LIN{ E6POS: X 712.0875, Y 3.2381, Z -130.0150, A 0, B 90, C 0, E1 0, E2 0, E3 0, E4 0 } C_DIS
LIN{ E6POS: X 712.0906, Y 3.3238, Z -130.0150, A 0, B 90, C 0, E1 0, E2 0, E3 0, E4 0 } C_DIS
LIN{ E6POS: X 712.1099, Y 3.6631, Z -130.0150, A 0, B 90, C 0, E1 0, E2 0, E3 0, E4 0 } C_DIS
LIN{ E6POS: X 712.1445, Y 4.6625, Z -130.0150, A 0, B 90, C 0, E1 0, E2 0, E3 0, E4 0 } C_DIS
LIN{ E6POS: X 712.1475, Y 4.7471, Z -130.0150, A 0, B 90, C 0, E1 0, E2 0, E3 0, E4 0 } C_DIS
LIN{ E6POS: X 712.1666, Y 5.0859, Z -130.0150, A 0, B 90, C 0, E1 0, E2 0, E3 0, E4 0 } C_DIS
LIN{ E6POS: X 712.2006, Y 6.0853, Z -130.0150, A 0, B 90, C 0, E1 0, E2 0, E3 0, E4 0 } C_DIS
LIN{ E6POS: X 712.2023, Y 6.1349, Z -130.0150, A 0, B 90, C 0, E1 0, E2 0, E3 0, E4 0 } C_DIS
LIN{ E6POS: X 712.2215, Y 6.4624, Z -130.0150, A 0, B 90, C 0, E1 0, E2 0, E3 0, E4 0 } C_DIS
LIN{ E6POS: X 712.2546, Y 7.4428, Z -130.0150, A 0, B 90, C 0, E1 0, E2 0, E3 0, E4 0 } C_DIS
LIN{ E6POS: X 712.2745, Y 7.7486, Z -130.0150, A 0, B 90, C 0, E1 0, E2 0, E3 0, E4 0 } C_DIS
LIN{ E6POS: X 712.3050, Y 8.6935, Z -130.0150, A 0, B 90, C 0, E1 0, E2 0, E3 0, E4 0 } C_DIS
LIN{ E6POS: X 712.3249, Y 8.9881, Z -130.0150, A 0, B 90, C 0, E1 0, E2 0, E3 0, E4 0 } C_DIS
LIN{ E6POS: X 712.3556, Y 9.9312, Z -130.0150, A 0, B 90, C 0, E1 0, E2 0, E3 0, E4 0 } C_DIS
LIN{ E6POS: X 712.3754, Y 10.2252, Z -130.0150, A 0, B 90, C 0, E1 0, E2 0, E3 0, E4 0 } C_DIS
LIN{ E6POS: X 712.4064, Y 11.1999, Z -130.0150, A 0, B 90, C 0, E1 0, E2 0, E3 0, E4 0 } C_DIS
LIN{ E6POS: X 712.4258, Y 11.5039, Z -130.0150, A 0, B 90, C 0, E1 0, E2 0, E3 0, E4 0 } C_DIS
LIN{ E6POS: X 712.4588, Y 12.5033, Z -130.0150, A 0, B 90, C 0, E1 0, E2 0, E3 0, E4 0 } C_DIS
LIN{ E6POS: X 712.4601, Y 12.5446, Z -130.0150, A 0, B 90, C 0, E1 0, E2 0, E3 0, E4 0 } C_DIS
LIN{ E6POS: X 712.4786, Y 12.8694, Z -130.0150, A 0, B 90, C 0, E1 0, E2 0, E3 0, E4 0 } C_DIS
LIN{ E6POS: X 712.5115, Y 13.8689, Z -130.0150, A 0, B 90, C 0, E1 0, E2 0, E3 0, E4 0 } C_DIS
LIN{ E6POS: X 712.5138, Y 13.9415, Z -130.0150, A 0, B 90, C 0, E1 0, E2 0, E3 0, E4 0 } C_DIS
LIN{ E6POS: X 712.5317, Y 14.2765, Z -130.0150, A 0, B 90, C 0, E1 0, E2 0, E3 0, E4 0 } C_DIS
LIN{ E6POS: X 712.5651, Y 15.2759, Z -130.0150, A 0, B 90, C 0, E1 0, E2 0, E3 0, E4 0 } C_DIS
LIN{ E6POS: X 712.5675, Y 15.3476, Z -130.0150, A 0, B 90, C 0, E1 0, E2 0, E3 0, E4 0 } C_DIS
LIN{ E6POS: X 712.5857, Y 15.6822, Z -130.0150, A 0, B 90, C 0, E1 0, E2 0, E3 0, E4 0 } C_DIS
LIN{ E6POS: X 712.6192, Y 16.6816, Z -130.0150, A 0, B 90, C 0, E1 0, E2 0, E3 0, E4 0 } C_DIS
LIN{ E6POS: X 712.6205, Y 16.7189, Z -130.0150, A 0, B 90, C 0, E1 0, E2 0, E3 0, E4 0 } C_DIS
LIN{ E6POS: X 712.6389, Y 17.0427, Z -130.0150, A 0, B 90, C 0, E1 0, E2 0, E3 0, E4 0 } C_DIS
LIN{ E6POS: X 712.6716, Y 18.0105, Z -130.0150, A 0, B 90, C 0, E1 0, E2 0, E3 0, E4 0 } C_DIS
LIN{ E6POS: X 712.6913, Y 18.3127, Z -130.0150, A 0, B 90, C 0, E1 0, E2 0, E3 0, E4 0 } C_DIS
LIN{ E6POS: X 712.7222, Y 19.2455, Z -130.0150, A 0, B 90, C 0, E1 0, E2 0, E3 0, E4 0 } C_DIS
LIN{ E6POS: X 712.7422, Y 19.5366, Z -130.0150, A 0, B 90, C 0, E1 0, E2 0, E3 0, E4 0 } C_DIS
LIN{ E6POS: X 712.7740, Y 20.4676, Z -130.0150, A 0, B 90, C 0, E1 0, E2 0, E3 0, E4 0 } C_DIS
LIN{ E6POS: X 712.7943, Y 20.7581, Z -130.0150, A 0, B 90, C 0, E1 0, E2 0, E3 0, E4 0 } C_DIS
LIN{ E6POS: X 712.8292, Y 21.7205, Z -130.0150, A 0, B 90, C 0, E1 0, E2 0, E3 0, E4 0 } C_DIS
LIN{ E6POS: X 712.8492, Y 22.0206, Z -130.0150, A 0, B 90, C 0, E1 0, E2 0, E3 0, E4 0 } C_DIS
LIN{ E6POS: X 712.8860, Y 23.0199, Z -130.0150, A 0, B 90, C 0, E1 0, E2 0, E3 0, E4 0 } C_DIS
LIN{ E6POS: X 712.8870, Y 23.0469, Z -130.0150, A 0, B 90, C 0, E1 0, E2 0, E3 0, E4 0 } C_DIS
LIN{ E6POS: X 712.9064, Y 23.3674, Z -130.0150, A 0, B 90, C 0, E1 0, E2 0, E3 0, E4 0 } C_DIS
LIN{ E6POS: X 712.9477, Y 24.3665, Z -130.0150, A 0, B 90, C 0, E1 0, E2 0, E3 0, E4 0 } C_DIS
LIN{ E6POS: X 712.9490, Y 24.3984, Z -130.0150, A 0, B 90, C 0, E1 0, E2 0, E3 0, E4 0 } C_DIS
LIN{ E6POS: X 712.9686, Y 24.7244, Z -130.0150, A 0, B 90, C 0, E1 0, E2 0, E3 0, E4 0 } C_DIS
LIN{ E6POS: X 713.0131, Y 25.6987, Z -130.0150, A 0, B 90, C 0, E1 0, E2 0, E3 0, E4 0 } C_DIS
LIN{ E6POS: X 713.0333, Y 26.0155, Z -130.0150, A 0, B 90, C 0, E1 0, E2 0, E3 0, E4 0 } C_DIS
LIN{ E6POS: X 713.1012, Y 27.0132, Z -130.0150, A 0, B 90, C 0, E1 0, E2 0, E3 0, E4 0 } C_DIS
LIN{ E6POS: X 713.1591, Y 27.8651, Z -130.0150, A 0, B 90, C 0, E1 0, E2 0, E3 0, E4 0 } C_DIS
LIN{ E6POS: X 713.1805, Y 28.1585, Z -130.0150, A 0, B 90, C 0, E1 0, E2 0, E3 0, E4 0 } C_DIS
LIN{ E6POS: X 713.2037, Y 28.4137, Z -130.0150, A 0, B 90, C 0, E1 0, E2 0, E3 0, E4 0 } C_DIS
LIN{ E6POS: X 713.2279, Y 28.6538, Z -130.0150, A 0, B 90, C 0, E1 0, E2 0, E3 0, E4 0 } C_DIS
LIN{ E6POS: X 713.2526, Y 28.9018, Z -130.0150, A 0, B 90, C 0, E1 0, E2 0, E3 0, E4 0 } C_DIS
LIN{ E6POS: X 713.3221, Y 29.8994, Z -130.0150, A 0, B 90, C 0, E1 0, E2 0, E3 0, E4 0 } C_DIS
LIN{ E6POS: X 713.3798, Y 30.7264, Z -130.0150, A 0, B 90, C 0, E1 0, E2 0, E3 0, E4 0 } C_DIS
LIN{ E6POS: X 713.4036, Y 31.0052, Z -130.0150, A 0, B 90, C 0, E1 0, E2 0, E3 0, E4 0 } C_DIS
LIN{ E6POS: X 713.4446, Y 32.0043, Z -130.0150, A 0, B 90, C 0, E1 0, E2 0, E3 0, E4 0 } C_DIS
LIN{ E6POS: X 713.4495, Y 32.1244, Z -130.0150, A 0, B 90, C 0, E1 0, E2 0, E3 0, E4 0 } C_DIS
LIN{ E6POS: X 713.4719, Y 32.4573, Z -130.0150, A 0, B 90, C 0, E1 0, E2 0, E3 0, E4 0 } C_DIS
LIN{ E6POS: X 713.5074, Y 33.4566, Z -130.0150, A 0, B 90, C 0, E1 0, E2 0, E3 0, E4 0 } C_DIS
LIN{ E6POS: X 713.5167, Y 33.7167, Z -130.0150, A 0, B 90, C 0, E1 0, E2 0, E3 0, E4 0 } C_DIS
LIN{ E6POS: X 713.5383, Y 34.0760, Z -130.0150, A 0, B 90, C 0, E1 0, E2 0, E3 0, E4 0 } C_DIS
LIN{ E6POS: X 713.5743, Y 35.0753, Z -130.0150, A 0, B 90, C 0, E1 0, E2 0, E3 0, E4 0 } C_DIS
LIN{ E6POS: X 713.5836, Y 35.3345, Z -130.0150, A 0, B 90, C 0, E1 0, E2 0, E3 0, E4 0 } C_DIS
LIN{ E6POS: X 713.6057, Y 35.6936, Z -130.0150, A 0, B 90, C 0, E1 0, E2 0, E3 0, E4 0 } C_DIS
LIN{ E6POS: X 713.6489, Y 36.6927, Z -130.0150, A 0, B 90, C 0, E1 0, E2 0, E3 0, E4 0 } C_DIS
LIN{ E6POS: X 713.6541, Y 36.8113, Z -130.0150, A 0, B 90, C 0, E1 0, E2 0, E3 0, E4 0 } C_DIS
LIN{ E6POS: X 713.6775, Y 37.1430, Z -130.0150, A 0, B 90, C 0, E1 0, E2 0, E3 0, E4 0 } C_DIS
LIN{ E6POS: X 713.7518, Y 38.1403, Z -130.0150, A 0, B 90, C 0, E1 0, E2 0, E3 0, E4 0 } C_DIS
LIN{ E6POS: X 713.7913, Y 38.6709, Z -130.0150, A 0, B 90, C 0, E1 0, E2 0, E3 0, E4 0 } C_DIS
LIN{ E6POS: X 713.8170, Y 38.9482, Z -130.0150, A 0, B 90, C 0, E1 0, E2 0, E3 0, E4 0 } C_DIS
LIN{ E6POS: X 713.8444, Y 39.1979, Z -130.0150, A 0, B 90, C 0, E1 0, E2 0, E3 0, E4 0 } C_DIS
LIN{ E6POS: X 713.8728, Y 39.4464, Z -130.0150, A 0, B 90, C 0, E1 0, E2 0, E3 0, E4 0 } C_DIS
LIN{ E6POS: X 713.9560, Y 40.4430, Z -130.0150, A 0, B 90, C 0, E1 0, E2 0, E3 0, E4 0 } C_DIS
LIN{ E6POS: X 713.9993, Y 40.9624, Z -130.0150, A 0, B 90, C 0, E1 0, E2 0, E3 0, E4 0 } C_DIS
LIN{ E6POS: X 714.0283, Y 41.2367, Z -130.0150, A 0, B 90, C 0, E1 0, E2 0, E3 0, E4 0 } C_DIS
LIN{ E6POS: X 714.0908, Y 42.2347, Z -130.0150, A 0, B 90, C 0, E1 0, E2 0, E3 0, E4 0 } C_DIS
LIN{ E6POS: X 714.0971, Y 42.3362, Z -130.0150, A 0, B 90, C 0, E1 0, E2 0, E3 0, E4 0 } C_DIS
LIN{ E6POS: X 714.1256, Y 42.6631, Z -130.0150, A 0, B 90, C 0, E1 0, E2 0, E3 0, E4 0 } C_DIS
LIN{ E6POS: X 714.1815, Y 43.6615, Z -130.0150, A 0, B 90, C 0, E1 0, E2 0, E3 0, E4 0 } C_DIS
LIN{ E6POS: X 714.1964, Y 43.9263, Z -130.0150, A 0, B 90, C 0, E1 0, E2 0, E3 0, E4 0 } C_DIS
LIN{ E6POS: X 714.2252, Y 44.2833, Z -130.0150, A 0, B 90, C 0, E1 0, E2 0, E3 0, E4 0 } C_DIS
LIN{ E6POS: X 714.2796, Y 45.2818, Z -130.0150, A 0, B 90, C 0, E1 0, E2 0, E3 0, E4 0 } C_DIS
LIN{ E6POS: X 714.2967, Y 45.5968, Z -130.0150, A 0, B 90, C 0, E1 0, E2 0, E3 0, E4 0 } C_DIS
LIN{ E6POS: X 714.3259, Y 45.9616, Z -130.0150, A 0, B 90, C 0, E1 0, E2 0, E3 0, E4 0 } C_DIS
LIN{ E6POS: X 714.3828, Y 46.9600, Z -130.0150, A 0, B 90, C 0, E1 0, E2 0, E3 0, E4 0 } C_DIS
LIN{ E6POS: X 714.3973, Y 47.2159, Z -130.0150, A 0, B 90, C 0, E1 0, E2 0, E3 0, E4 0 } C_DIS
LIN{ E6POS: X 714.4272, Y 47.5666, Z -130.0150, A 0, B 90, C 0, E1 0, E2 0, E3 0, E4 0 } C_DIS
LIN{ E6POS: X 714.4923, Y 48.5645, Z -130.0150, A 0, B 90, C 0, E1 0, E2 0, E3 0, E4 0 } C_DIS
LIN{ E6POS: X 714.4978, Y 48.6481, Z -130.0150, A 0, B 90, C 0, E1 0, E2 0, E3 0, E4 0 } C_DIS
LIN{ E6POS: X 714.5287, Y 48.9623, Z -130.0150, A 0, B 90, C 0, E1 0, E2 0, E3 0, E4 0 } C_DIS
LIN{ E6POS: X 714.5991, Y 49.9151, Z -130.0150, A 0, B 90, C 0, E1 0, E2 0, E3 0, E4 0 } C_DIS
LIN{ E6POS: X 714.6305, Y 50.2017, Z -130.0150, A 0, B 90, C 0, E1 0, E2 0, E3 0, E4 0 } C_DIS
LIN{ E6POS: X 714.7003, Y 51.0686, Z -130.0150, A 0, B 90, C 0, E1 0, E2 0, E3 0, E4 0 } C_DIS
LIN{ E6POS: X 714.7325, Y 51.3369, Z -130.0150, A 0, B 90, C 0, E1 0, E2 0, E3 0, E4 0 } C_DIS
LIN{ E6POS: X 714.8029, Y 52.1697, Z -130.0150, A 0, B 90, C 0, E1 0, E2 0, E3 0, E4 0 } C_DIS
LIN{ E6POS: X 714.8884, Y 52.4223, Z -130.0150, A 0, B 90, C 0, E1 0, E2 0, E3 0, E4 0 } C_DIS
LIN{ E6POS: X 715.6198, Y 52.2627, Z -130.0150, A 0, B 90, C 0, E1 0, E2 0, E3 0, E4 0 } C_DIS
LIN{ E6POS: X 716.5857, Y 52.0038, Z -130.0150, A 0, B 90, C 0, E1 0, E2 0, E3 0, E4 0 } C_DIS
LIN{ E6POS: X 717.5516, Y 51.7450, Z -130.0150, A 0, B 90, C 0, E1 0, E2 0, E3 0, E4 0 } C_DIS
LIN{ E6POS: X 717.8004, Y 51.6783, Z -130.0150, A 0, B 90, C 0, E1 0, E2 0, E3 0, E4 0 } C_DIS
LIN{ E6POS: X 718.5842, Y 51.4709, Z -130.0150, A 0, B 90, C 0, E1 0, E2 0, E3 0, E4 0 } C_DIS
LIN{ E6POS: X 719.5486, Y 51.2064, Z -130.0150, A 0, B 90, C 0, E1 0, E2 0, E3 0, E4 0 } C_DIS
LIN{ E6POS: X 720.5129, Y 50.9418, Z -130.0150, A 0, B 90, C 0, E1 0, E2 0, E3 0, E4 0 } C_DIS
LIN{ E6POS: X 721.4773, Y 50.6773, Z -130.0150, A 0, B 90, C 0, E1 0, E2 0, E3 0, E4 0 } C_DIS
LIN{ E6POS: X 722.4417, Y 50.4127, Z -130.0150, A 0, B 90, C 0, E1 0, E2 0, E3 0, E4 0 } C_DIS
LIN{ E6POS: X 722.9421, Y 50.2755, Z -130.0150, A 0, B 90, C 0, E1 0, E2 0, E3 0, E4 0 } C_DIS
LIN{ E6POS: X 723.9022, Y 49.9957, Z -130.0150, A 0, B 90, C 0, E1 0, E2 0, E3 0, E4 0 } C_DIS
LIN{ E6POS: X 724.1924, Y 49.9112, Z -130.0150, A 0, B 90, C 0, E1 0, E2 0, E3 0, E4 0 } C_DIS
LIN{ E6POS: X 725.1562, Y 49.6446, Z -130.0150, A 0, B 90, C 0, E1 0, E2 0, E3 0, E4 0 } C_DIS
LIN{ E6POS: X 726.1200, Y 49.3780, Z -130.0150, A 0, B 90, C 0, E1 0, E2 0, E3 0, E4 0 } C_DIS
LIN{ E6POS: X 727.0838, Y 49.1113, Z -130.0150, A 0, B 90, C 0, E1 0, E2 0, E3 0, E4 0 } C_DIS
LIN{ E6POS: X 728.0476, Y 48.8447, Z -130.0150, A 0, B 90, C 0, E1 0, E2 0, E3 0, E4 0 } C_DIS
LIN{ E6POS: X 729.0114, Y 48.5781, Z -130.0150, A 0, B 90, C 0, E1 0, E2 0, E3 0, E4 0 } C_DIS
LIN{ E6POS: X 729.9752, Y 48.3115, Z -130.0150, A 0, B 90, C 0, E1 0, E2 0, E3 0, E4 0 } C_DIS
LIN{ E6POS: X 730.9390, Y 48.0449, Z -130.0150, A 0, B 90, C 0, E1 0, E2 0, E3 0, E4 0 } C_DIS
LIN{ E6POS: X 731.4545, Y 47.9023, Z -130.0150, A 0, B 90, C 0, E1 0, E2 0, E3 0, E4 0 } C_DIS
LIN{ E6POS: X 732.4135, Y 47.6189, Z -130.0150, A 0, B 90, C 0, E1 0, E2 0, E3 0, E4 0 } C_DIS
LIN{ E6POS: X 733.3725, Y 47.3356, Z -130.0150, A 0, B 90, C 0, E1 0, E2 0, E3 0, E4 0 } C_DIS
LIN{ E6POS: X 733.5370, Y 47.2870, Z -130.0150, A 0, B 90, C 0, E1 0, E2 0, E3 0, E4 0 } C_DIS
LIN{ E6POS: X 734.5038, Y 47.0312, Z -130.0150, A 0, B 90, C 0, E1 0, E2 0, E3 0, E4 0 } C_DIS
LIN{ E6POS: X 735.4705, Y 46.7755, Z -130.0150, A 0, B 90, C 0, E1 0, E2 0, E3 0, E4 0 } C_DIS
LIN{ E6POS: X 736.4372, Y 46.5197, Z -130.0150, A 0, B 90, C 0, E1 0, E2 0, E3 0, E4 0 } C_DIS
LIN{ E6POS: X 737.4040, Y 46.2639, Z -130.0150, A 0, B 90, C 0, E1 0, E2 0, E3 0, E4 0 } C_DIS
LIN{ E6POS: X 738.3707, Y 46.0082, Z -130.0150, A 0, B 90, C 0, E1 0, E2 0, E3 0, E4 0 } C_DIS
LIN{ E6POS: X 739.3374, Y 45.7524, Z -130.0150, A 0, B 90, C 0, E1 0, E2 0, E3 0, E4 0 } C_DIS
LIN{ E6POS: X 740.3042, Y 45.4966, Z -130.0150, A 0, B 90, C 0, E1 0, E2 0, E3 0, E4 0 } C_DIS
LIN{ E6POS: X 741.2709, Y 45.2409, Z -130.0150, A 0, B 90, C 0, E1 0, E2 0, E3 0, E4 0 } C_DIS
LIN{ E6POS: X 742.2377, Y 44.9851, Z -130.0150, A 0, B 90, C 0, E1 0, E2 0, E3 0, E4 0 } C_DIS
LIN{ E6POS: X 742.5361, Y 44.9061, Z -130.0150, A 0, B 90, C 0, E1 0, E2 0, E3 0, E4 0 } C_DIS
LIN{ E6POS: X 743.4986, Y 44.6349, Z -130.0150, A 0, B 90, C 0, E1 0, E2 0, E3 0, E4 0 } C_DIS
LIN{ E6POS: X 744.4611, Y 44.3637, Z -130.0150, A 0, B 90, C 0, E1 0, E2 0, E3 0, E4 0 } C_DIS
LIN{ E6POS: X 745.1256, Y 44.1764, Z -130.0150, A 0, B 90, C 0, E1 0, E2 0, E3 0, E4 0 } C_DIS
LIN{ E6POS: X 746.0978, Y 43.9420, Z -130.0150, A 0, B 90, C 0, E1 0, E2 0, E3 0, E4 0 } C_DIS
LIN{ E6POS: X 747.0699, Y 43.7075, Z -130.0150, A 0, B 90, C 0, E1 0, E2 0, E3 0, E4 0 } C_DIS
LIN{ E6POS: X 748.0420, Y 43.4731, Z -130.0150, A 0, B 90, C 0, E1 0, E2 0, E3 0, E4 0 } C_DIS
LIN{ E6POS: X 749.0142, Y 43.2386, Z -130.0150, A 0, B 90, C 0, E1 0, E2 0, E3 0, E4 0 } C_DIS
LIN{ E6POS: X 749.9863, Y 43.0042, Z -130.0150, A 0, B 90, C 0, E1 0, E2 0, E3 0, E4 0 } C_DIS
LIN{ E6POS: X 750.9584, Y 42.7697, Z -130.0150, A 0, B 90, C 0, E1 0, E2 0, E3 0, E4 0 } C_DIS
LIN{ E6POS: X 751.9305, Y 42.5353, Z -130.0150, A 0, B 90, C 0, E1 0, E2 0, E3 0, E4 0 } C_DIS
LIN{ E6POS: X 752.9027, Y 42.3008, Z -130.0150, A 0, B 90, C 0, E1 0, E2 0, E3 0, E4 0 } C_DIS
LIN{ E6POS: X 753.8748, Y 42.0664, Z -130.0150, A 0, B 90, C 0, E1 0, E2 0, E3 0, E4 0 } C_DIS
LIN{ E6POS: X 754.6995, Y 41.8675, Z -130.0150, A 0, B 90, C 0, E1 0, E2 0, E3 0, E4 0 } C_DIS
LIN{ E6POS: X 755.6683, Y 41.6200, Z -130.0150, A 0, B 90, C 0, E1 0, E2 0, E3 0, E4 0 } C_DIS
LIN{ E6POS: X 756.6372, Y 41.3724, Z -130.0150, A 0, B 90, C 0, E1 0, E2 0, E3 0, E4 0 } C_DIS
LIN{ E6POS: X 757.4699, Y 41.1597, Z -130.0150, A 0, B 90, C 0, E1 0, E2 0, E3 0, E4 0 } C_DIS
LIN{ E6POS: X 758.4505, Y 40.9637, Z -130.0150, A 0, B 90, C 0, E1 0, E2 0, E3 0, E4 0 } C_DIS
LIN{ E6POS: X 759.4311, Y 40.7676, Z -130.0150, A 0, B 90, C 0, E1 0, E2 0, E3 0, E4 0 } C_DIS
LIN{ E6POS: X 760.4117, Y 40.5716, Z -130.0150, A 0, B 90, C 0, E1 0, E2 0, E3 0, E4 0 } C_DIS
LIN{ E6POS: X 761.3923, Y 40.3756, Z -130.0150, A 0, B 90, C 0, E1 0, E2 0, E3 0, E4 0 } C_DIS
LIN{ E6POS: X 762.3729, Y 40.1795, Z -130.0150, A 0, B 90, C 0, E1 0, E2 0, E3 0, E4 0 } C_DIS
LIN{ E6POS: X 763.3535, Y 39.9835, Z -130.0150, A 0, B 90, C 0, E1 0, E2 0, E3 0, E4 0 } C_DIS
LIN{ E6POS: X 764.3340, Y 39.7875, Z -130.0150, A 0, B 90, C 0, E1 0, E2 0, E3 0, E4 0 } C_DIS
LIN{ E6POS: X 765.3146, Y 39.5914, Z -130.0150, A 0, B 90, C 0, E1 0, E2 0, E3 0, E4 0 } C_DIS
LIN{ E6POS: X 766.2952, Y 39.3954, Z -130.0150, A 0, B 90, C 0, E1 0, E2 0, E3 0, E4 0 } C_DIS
LIN{ E6POS: X 766.4520, Y 39.3641, Z -130.0150, A 0, B 90, C 0, E1 0, E2 0, E3 0, E4 0 } C_DIS
LIN{ E6POS: X 767.4308, Y 39.1593, Z -130.0150, A 0, B 90, C 0, E1 0, E2 0, E3 0, E4 0 } C_DIS
LIN{ E6POS: X 768.4096, Y 38.9546, Z -130.0150, A 0, B 90, C 0, E1 0, E2 0, E3 0, E4 0 } C_DIS
LIN{ E6POS: X 769.0778, Y 38.8148, Z -130.0150, A 0, B 90, C 0, E1 0, E2 0, E3 0, E4 0 } C_DIS
LIN{ E6POS: X 770.0711, Y 38.6997, Z -130.0150, A 0, B 90, C 0, E1 0, E2 0, E3 0, E4 0 } C_DIS
LIN{ E6POS: X 771.0645, Y 38.5845, Z -130.0150, A 0, B 90, C 0, E1 0, E2 0, E3 0, E4 0 } C_DIS
LIN{ E6POS: X 772.0578, Y 38.4693, Z -130.0150, A 0, B 90, C 0, E1 0, E2 0, E3 0, E4 0 } C_DIS
LIN{ E6POS: X 773.0512, Y 38.3542, Z -130.0150, A 0, B 90, C 0, E1 0, E2 0, E3 0, E4 0 } C_DIS
LIN{ E6POS: X 774.0445, Y 38.2390, Z -130.0150, A 0, B 90, C 0, E1 0, E2 0, E3 0, E4 0 } C_DIS
LIN{ E6POS: X 775.0379, Y 38.1239, Z -130.0150, A 0, B 90, C 0, E1 0, E2 0, E3 0, E4 0 } C_DIS
LIN{ E6POS: X 776.0312, Y 38.0087, Z -130.0150, A 0, B 90, C 0, E1 0, E2 0, E3 0, E4 0 } C_DIS
LIN{ E6POS: X 776.3033, Y 37.9772, Z -130.0150, A 0, B 90, C 0, E1 0, E2 0, E3 0, E4 0 } C_DIS
LIN{ E6POS: X 777.2964, Y 37.8600, Z -130.0150, A 0, B 90, C 0, E1 0, E2 0, E3 0, E4 0 } C_DIS
LIN{ E6POS: X 778.2895, Y 37.7429, Z -130.0150, A 0, B 90, C 0, E1 0, E2 0, E3 0, E4 0 } C_DIS
LIN{ E6POS: X 778.4588, Y 37.7230, Z -130.0150, A 0, B 90, C 0, E1 0, E2 0, E3 0, E4 0 } C_DIS
LIN{ E6POS: X 779.4586, Y 37.7025, Z -130.0150, A 0, B 90, C 0, E1 0, E2 0, E3 0, E4 0 } C_DIS
LIN{ E6POS: X 780.4584, Y 37.6820, Z -130.0150, A 0, B 90, C 0, E1 0, E2 0, E3 0, E4 0 } C_DIS
LIN{ E6POS: X 781.4582, Y 37.6616, Z -130.0150, A 0, B 90, C 0, E1 0, E2 0, E3 0, E4 0 } C_DIS
LIN{ E6POS: X 782.4579, Y 37.6411, Z -130.0150, A 0, B 90, C 0, E1 0, E2 0, E3 0, E4 0 } C_DIS
LIN{ E6POS: X 783.4577, Y 37.6206, Z -130.0150, A 0, B 90, C 0, E1 0, E2 0, E3 0, E4 0 } C_DIS
LIN{ E6POS: X 784.3674, Y 37.6020, Z -130.0150, A 0, B 90, C 0, E1 0, E2 0, E3 0, E4 0 } C_DIS
LIN{ E6POS: X 785.3672, Y 37.5838, Z -130.0150, A 0, B 90, C 0, E1 0, E2 0, E3 0, E4 0 } C_DIS
LIN{ E6POS: X 786.1700, Y 37.5692, Z -130.0150, A 0, B 90, C 0, E1 0, E2 0, E3 0, E4 0 } C_DIS
LIN{ E6POS: X 787.1675, Y 37.6400, Z -130.0150, A 0, B 90, C 0, E1 0, E2 0, E3 0, E4 0 } C_DIS
LIN{ E6POS: X 788.1650, Y 37.7108, Z -130.0150, A 0, B 90, C 0, E1 0, E2 0, E3 0, E4 0 } C_DIS
LIN{ E6POS: X 789.1625, Y 37.7816, Z -130.0150, A 0, B 90, C 0, E1 0, E2 0, E3 0, E4 0 } C_DIS
LIN{ E6POS: X 790.1600, Y 37.8524, Z -130.0150, A 0, B 90, C 0, E1 0, E2 0, E3 0, E4 0 } C_DIS
LIN{ E6POS: X 791.1575, Y 37.9232, Z -130.0150, A 0, B 90, C 0, E1 0, E2 0, E3 0, E4 0 } C_DIS
LIN{ E6POS: X 791.2008, Y 37.9263, Z -130.0150, A 0, B 90, C 0, E1 0, E2 0, E3 0, E4 0 } C_DIS
LIN{ E6POS: X 792.1981, Y 37.9992, Z -130.0150, A 0, B 90, C 0, E1 0, E2 0, E3 0, E4 0 } C_DIS
LIN{ E6POS: X 792.7685, Y 38.0409, Z -130.0150, A 0, B 90, C 0, E1 0, E2 0, E3 0, E4 0 } C_DIS
LIN{ E6POS: X 793.7601, Y 38.1698, Z -130.0150, A 0, B 90, C 0, E1 0, E2 0, E3 0, E4 0 } C_DIS
LIN{ E6POS: X 794.7518, Y 38.2986, Z -130.0150, A 0, B 90, C 0, E1 0, E2 0, E3 0, E4 0 } C_DIS
LIN{ E6POS: X 795.7435, Y 38.4275, Z -130.0150, A 0, B 90, C 0, E1 0, E2 0, E3 0, E4 0 } C_DIS
LIN{ E6POS: X 796.7351, Y 38.5564, Z -130.0150, A 0, B 90, C 0, E1 0, E2 0, E3 0, E4 0 } C_DIS
LIN{ E6POS: X 797.3598, Y 38.6376, Z -130.0150, A 0, B 90, C 0, E1 0, E2 0, E3 0, E4 0 } C_DIS
LIN{ E6POS: X 798.3514, Y 38.7665, Z -130.0150, A 0, B 90, C 0, E1 0, E2 0, E3 0, E4 0 } C_DIS
LIN{ E6POS: X 798.8097, Y 38.8260, Z -130.0150, A 0, B 90, C 0, E1 0, E2 0, E3 0, E4 0 } C_DIS
LIN{ E6POS: X 798.7068, Y 37.8313, Z -130.0150, A 0, B 90, C 0, E1 0, E2 0, E3 0, E4 0 } C_DIS
LIN{ E6POS: X 798.6040, Y 36.8366, Z -130.0150, A 0, B 90, C 0, E1 0, E2 0, E3 0, E4 0 } C_DIS
LIN{ E6POS: X 798.5012, Y 35.8419, Z -130.0150, A 0, B 90, C 0, E1 0, E2 0, E3 0, E4 0 } C_DIS
LIN{ E6POS: X 798.3983, Y 34.8472, Z -130.0150, A 0, B 90, C 0, E1 0, E2 0, E3 0, E4 0 } C_DIS
LIN{ E6POS: X 798.2955, Y 33.8525, Z -130.0150, A 0, B 90, C 0, E1 0, E2 0, E3 0, E4 0 } C_DIS
LIN{ E6POS: X 798.1927, Y 32.8578, Z -130.0150, A 0, B 90, C 0, E1 0, E2 0, E3 0, E4 0 } C_DIS
LIN{ E6POS: X 798.0898, Y 31.8631, Z -130.0150, A 0, B 90, C 0, E1 0, E2 0, E3 0, E4 0 } C_DIS
LIN{ E6POS: X 797.9870, Y 30.8684, Z -130.0150, A 0, B 90, C 0, E1 0, E2 0, E3 0, E4 0 } C_DIS
LIN{ E6POS: X 797.8842, Y 29.8737, Z -130.0150, A 0, B 90, C 0, E1 0, E2 0, E3 0, E4 0 } C_DIS
LIN{ E6POS: X 797.7813, Y 28.8790, Z -130.0150, A 0, B 90, C 0, E1 0, E2 0, E3 0, E4 0 } C_DIS
LIN{ E6POS: X 797.6785, Y 27.8843, Z -130.0150, A 0, B 90, C 0, E1 0, E2 0, E3 0, E4 0 } C_DIS
LIN{ E6POS: X 797.5757, Y 26.8896, Z -130.0150, A 0, B 90, C 0, E1 0, E2 0, E3 0, E4 0 } C_DIS
LIN{ E6POS: X 797.5273, Y 26.4221, Z -130.0150, A 0, B 90, C 0, E1 0, E2 0, E3 0, E4 0 } C_DIS
LIN{ E6POS: X 797.4245, Y 25.4274, Z -130.0150, A 0, B 90, C 0, E1 0, E2 0, E3 0, E4 0 } C_DIS
LIN{ E6POS: X 797.3217, Y 24.4327, Z -130.0150, A 0, B 90, C 0, E1 0, E2 0, E3 0, E4 0 } C_DIS
LIN{ E6POS: X 797.2188, Y 23.4380, Z -130.0150, A 0, B 90, C 0, E1 0, E2 0, E3 0, E4 0 } C_DIS
LIN{ E6POS: X 797.1224, Y 22.5051, Z -130.0150, A 0, B 90, C 0, E1 0, E2 0, E3 0, E4 0 } C_DIS
LIN{ E6POS: X 797.0002, Y 21.5126, Z -130.0150, A 0, B 90, C 0, E1 0, E2 0, E3 0, E4 0 } C_DIS
LIN{ E6POS: X 796.8780, Y 20.5201, Z -130.0150, A 0, B 90, C 0, E1 0, E2 0, E3 0, E4 0 } C_DIS
LIN{ E6POS: X 796.7559, Y 19.5276, Z -130.0150, A 0, B 90, C 0, E1 0, E2 0, E3 0, E4 0 } C_DIS
LIN{ E6POS: X 796.6337, Y 18.5351, Z -130.0150, A 0, B 90, C 0, E1 0, E2 0, E3 0, E4 0 } C_DIS
LIN{ E6POS: X 796.5115, Y 17.5426, Z -130.0150, A 0, B 90, C 0, E1 0, E2 0, E3 0, E4 0 } C_DIS
LIN{ E6POS: X 796.3893, Y 16.5500, Z -130.0150, A 0, B 90, C 0, E1 0, E2 0, E3 0, E4 0 } C_DIS
LIN{ E6POS: X 796.2672, Y 15.5575, Z -130.0150, A 0, B 90, C 0, E1 0, E2 0, E3 0, E4 0 } C_DIS
LIN{ E6POS: X 796.1450, Y 14.5650, Z -130.0150, A 0, B 90, C 0, E1 0, E2 0, E3 0, E4 0 } C_DIS
LIN{ E6POS: X 796.0228, Y 13.5725, Z -130.0150, A 0, B 90, C 0, E1 0, E2 0, E3 0, E4 0 } C_DIS
LIN{ E6POS: X 795.9006, Y 12.5800, Z -130.0150, A 0, B 90, C 0, E1 0, E2 0, E3 0, E4 0 } C_DIS
LIN{ E6POS: X 795.7785, Y 11.5875, Z -130.0150, A 0, B 90, C 0, E1 0, E2 0, E3 0, E4 0 } C_DIS
LIN{ E6POS: X 795.7041, Y 10.9836, Z -130.0150, A 0, B 90, C 0, E1 0, E2 0, E3 0, E4 0 } C_DIS
LIN{ E6POS: X 795.5819, Y 9.9911, Z -130.0150, A 0, B 90, C 0, E1 0, E2 0, E3 0, E4 0 } C_DIS
LIN{ E6POS: X 795.4598, Y 8.9986, Z -130.0150, A 0, B 90, C 0, E1 0, E2 0, E3 0, E4 0 } C_DIS
LIN{ E6POS: X 795.3376, Y 8.0061, Z -130.0150, A 0, B 90, C 0, E1 0, E2 0, E3 0, E4 0 } C_DIS
LIN{ E6POS: X 795.2562, Y 7.3452, Z -128.0150, A 0, B 90, C 0, E1 0, E2 0, E3 0, E4 0 } C_DIS
LIN{ E6POS: X 795.0854, Y 6.3599, Z -128.0150, A 0, B 90, C 0, E1 0, E2 0, E3 0, E4 0 } C_DIS
LIN{ E6POS: X 794.9146, Y 5.3746, Z -128.0150, A 0, B 90, C 0, E1 0, E2 0, E3 0, E4 0 } C_DIS
LIN{ E6POS: X 794.7438, Y 4.3893, Z -128.0150, A 0, B 90, C 0, E1 0, E2 0, E3 0, E4 0 } C_DIS
LIN{ E6POS: X 794.5730, Y 3.4040, Z -128.0150, A 0, B 90, C 0, E1 0, E2 0, E3 0, E4 0 } C_DIS
LIN{ E6POS: X 794.4021, Y 2.4187, Z -128.0150, A 0, B 90, C 0, E1 0, E2 0, E3 0, E4 0 } C_DIS
LIN{ E6POS: X 794.2313, Y 1.4334, Z -128.0150, A 0, B 90, C 0, E1 0, E2 0, E3 0, E4 0 } C_DIS
LIN{ E6POS: X 794.0605, Y 0.4481, Z -128.0150, A 0, B 90, C 0, E1 0, E2 0, E3 0, E4 0 } C_DIS
LIN{ E6POS: X 793.8897, Y -0.5372, Z -128.0150, A 0, B 90, C 0, E1 0, E2 0, E3 0, E4 0 } C_DIS
LIN{ E6POS: X 793.7189, Y -1.5225, Z -128.0150, A 0, B 90, C 0, E1 0, E2 0, E3 0, E4 0 } C_DIS
LIN{ E6POS: X 793.5481, Y -2.5078, Z -128.0150, A 0, B 90, C 0, E1 0, E2 0, E3 0, E4 0 } C_DIS
LIN{ E6POS: X 793.3871, Y -3.4364, Z -128.0150, A 0, B 90, C 0, E1 0, E2 0, E3 0, E4 0 } C_DIS
LIN{ E6POS: X 793.2162, Y -4.4217, Z -128.0150, A 0, B 90, C 0, E1 0, E2 0, E3 0, E4 0 } C_DIS
LIN{ E6POS: X 793.0454, Y -5.4070, Z -128.0150, A 0, B 90, C 0, E1 0, E2 0, E3 0, E4 0 } C_DIS
LIN{ E6POS: X 793.0310, Y -5.4900, Z -128.0150, A 0, B 90, C 0, E1 0, E2 0, E3 0, E4 0 } C_DIS
LIN{ E6POS: X 792.7476, Y -6.4490, Z -128.0150, A 0, B 90, C 0, E1 0, E2 0, E3 0, E4 0 } C_DIS
LIN{ E6POS: X 792.4642, Y -7.4080, Z -128.0150, A 0, B 90, C 0, E1 0, E2 0, E3 0, E4 0 } C_DIS
LIN{ E6POS: X 792.1808, Y -8.3670, Z -128.0150, A 0, B 90, C 0, E1 0, E2 0, E3 0, E4 0 } C_DIS
LIN{ E6POS: X 791.8974, Y -9.3260, Z -128.0150, A 0, B 90, C 0, E1 0, E2 0, E3 0, E4 0 } C_DIS
LIN{ E6POS: X 791.6139, Y -10.2850, Z -128.0150, A 0, B 90, C 0, E1 0, E2 0, E3 0, E4 0 } C_DIS
LIN{ E6POS: X 791.3305, Y -11.2440, Z -128.0150, A 0, B 90, C 0, E1 0, E2 0, E3 0, E4 0 } C_DIS
LIN{ E6POS: X 791.0471, Y -12.2030, Z -128.0150, A 0, B 90, C 0, E1 0, E2 0, E3 0, E4 0 } C_DIS
LIN{ E6POS: X 790.7637, Y -13.1620, Z -128.0150, A 0, B 90, C 0, E1 0, E2 0, E3 0, E4 0 } C_DIS
LIN{ E6POS: X 790.7102, Y -13.3429, Z -128.0150, A 0, B 90, C 0, E1 0, E2 0, E3 0, E4 0 } C_DIS
LIN{ E6POS: X 790.4268, Y -14.3019, Z -128.0150, A 0, B 90, C 0, E1 0, E2 0, E3 0, E4 0 } C_DIS
LIN{ E6POS: X 790.2681, Y -14.8387, Z -128.0150, A 0, B 90, C 0, E1 0, E2 0, E3 0, E4 0 } C_DIS
LIN{ E6POS: X 789.6733, Y -15.6426, Z -128.0150, A 0, B 90, C 0, E1 0, E2 0, E3 0, E4 0 } C_DIS
LIN{ E6POS: X 789.0784, Y -16.4464, Z -128.0150, A 0, B 90, C 0, E1 0, E2 0, E3 0, E4 0 } C_DIS
LIN{ E6POS: X 788.4835, Y -17.2502, Z -128.0150, A 0, B 90, C 0, E1 0, E2 0, E3 0, E4 0 } C_DIS
LIN{ E6POS: X 787.8887, Y -18.0540, Z -128.0150, A 0, B 90, C 0, E1 0, E2 0, E3 0, E4 0 } C_DIS
LIN{ E6POS: X 787.3452, Y -18.7884, Z -128.0150, A 0, B 90, C 0, E1 0, E2 0, E3 0, E4 0 } C_DIS
LIN{ E6POS: X 786.7884, Y -19.5408, Z -128.0150, A 0, B 90, C 0, E1 0, E2 0, E3 0, E4 0 } C_DIS
LIN{ E6POS: X 785.8324, Y -19.8339, Z -128.0150, A 0, B 90, C 0, E1 0, E2 0, E3 0, E4 0 } C_DIS
LIN{ E6POS: X 784.8763, Y -20.1271, Z -128.0150, A 0, B 90, C 0, E1 0, E2 0, E3 0, E4 0 } C_DIS
LIN{ E6POS: X 783.9202, Y -20.4202, Z -128.0150, A 0, B 90, C 0, E1 0, E2 0, E3 0, E4 0 } C_DIS
LIN{ E6POS: X 783.1205, Y -20.6654, Z -128.0150, A 0, B 90, C 0, E1 0, E2 0, E3 0, E4 0 } C_DIS
LIN{ E6POS: X 782.4311, Y -20.8799, Z -128.0150, A 0, B 90, C 0, E1 0, E2 0, E3 0, E4 0 } C_DIS
LIN{ E6POS: X 781.5918, Y -20.7628, Z -128.0150, A 0, B 90, C 0, E1 0, E2 0, E3 0, E4 0 } C_DIS
LIN{ E6POS: X 780.6009, Y -20.6279, Z -128.0150, A 0, B 90, C 0, E1 0, E2 0, E3 0, E4 0 } C_DIS
LIN{ E6POS: X 779.6100, Y -20.4930, Z -128.0150, A 0, B 90, C 0, E1 0, E2 0, E3 0, E4 0 } C_DIS
LIN{ E6POS: X 778.6192, Y -20.3581, Z -128.0150, A 0, B 90, C 0, E1 0, E2 0, E3 0, E4 0 } C_DIS
LIN{ E6POS: X 777.6283, Y -20.2232, Z -128.0150, A 0, B 90, C 0, E1 0, E2 0, E3 0, E4 0 } C_DIS
LIN{ E6POS: X 777.0370, Y -20.1427, Z -128.0150, A 0, B 90, C 0, E1 0, E2 0, E3 0, E4 0 } C_DIS
LIN{ E6POS: X 776.0649, Y -19.9082, Z -128.0150, A 0, B 90, C 0, E1 0, E2 0, E3 0, E4 0 } C_DIS
LIN{ E6POS: X 776.0296, Y -19.8997, Z -128.0150, A 0, B 90, C 0, E1 0, E2 0, E3 0, E4 0 } C_DIS
LIN{ E6POS: X 775.0551, Y -19.6756, Z -128.0150, A 0, B 90, C 0, E1 0, E2 0, E3 0, E4 0 } C_DIS
LIN{ E6POS: X 774.0805, Y -19.4515, Z -128.0150, A 0, B 90, C 0, E1 0, E2 0, E3 0, E4 0 } C_DIS
LIN{ E6POS: X 773.1059, Y -19.2274, Z -128.0150, A 0, B 90, C 0, E1 0, E2 0, E3 0, E4 0 } C_DIS
LIN{ E6POS: X 772.1313, Y -19.0034, Z -128.0150, A 0, B 90, C 0, E1 0, E2 0, E3 0, E4 0 } C_DIS
LIN{ E6POS: X 771.1568, Y -18.7793, Z -128.0150, A 0, B 90, C 0, E1 0, E2 0, E3 0, E4 0 } C_DIS
LIN{ E6POS: X 770.4461, Y -18.6159, Z -128.0150, A 0, B 90, C 0, E1 0, E2 0, E3 0, E4 0 } C_DIS
LIN{ E6POS: X 769.4553, Y -18.4806, Z -128.0150, A 0, B 90, C 0, E1 0, E2 0, E3 0, E4 0 } C_DIS
LIN{ E6POS: X 769.2531, Y -18.4530, Z -128.0150, A 0, B 90, C 0, E1 0, E2 0, E3 0, E4 0 } C_DIS
LIN{ E6POS: X 768.2612, Y -18.3253, Z -128.0150, A 0, B 90, C 0, E1 0, E2 0, E3 0, E4 0 } C_DIS
LIN{ E6POS: X 767.2694, Y -18.1977, Z -128.0150, A 0, B 90, C 0, E1 0, E2 0, E3 0, E4 0 } C_DIS
LIN{ E6POS: X 766.2776, Y -18.0700, Z -128.0150, A 0, B 90, C 0, E1 0, E2 0, E3 0, E4 0 } C_DIS
LIN{ E6POS: X 765.2858, Y -17.9424, Z -128.0150, A 0, B 90, C 0, E1 0, E2 0, E3 0, E4 0 } C_DIS
LIN{ E6POS: X 764.2940, Y -17.8147, Z -128.0150, A 0, B 90, C 0, E1 0, E2 0, E3 0, E4 0 } C_DIS
LIN{ E6POS: X 763.3021, Y -17.6871, Z -128.0150, A 0, B 90, C 0, E1 0, E2 0, E3 0, E4 0 } C_DIS
LIN{ E6POS: X 762.4979, Y -17.5836, Z -128.0150, A 0, B 90, C 0, E1 0, E2 0, E3 0, E4 0 } C_DIS
LIN{ E6POS: X 761.5004, Y -17.5138, Z -128.0150, A 0, B 90, C 0, E1 0, E2 0, E3 0, E4 0 } C_DIS
LIN{ E6POS: X 761.2573, Y -17.4968, Z -128.0150, A 0, B 90, C 0, E1 0, E2 0, E3 0, E4 0 } C_DIS
LIN{ E6POS: X 760.2595, Y -17.4296, Z -128.0150, A 0, B 90, C 0, E1 0, E2 0, E3 0, E4 0 } C_DIS
LIN{ E6POS: X 759.2618, Y -17.3625, Z -128.0150, A 0, B 90, C 0, E1 0, E2 0, E3 0, E4 0 } C_DIS
LIN{ E6POS: X 758.2640, Y -17.2954, Z -128.0150, A 0, B 90, C 0, E1 0, E2 0, E3 0, E4 0 } C_DIS
LIN{ E6POS: X 757.2663, Y -17.2283, Z -128.0150, A 0, B 90, C 0, E1 0, E2 0, E3 0, E4 0 } C_DIS
LIN{ E6POS: X 756.2685, Y -17.1612, Z -128.0150, A 0, B 90, C 0, E1 0, E2 0, E3 0, E4 0 } C_DIS
LIN{ E6POS: X 755.2708, Y -17.0941, Z -128.0150, A 0, B 90, C 0, E1 0, E2 0, E3 0, E4 0 } C_DIS
LIN{ E6POS: X 754.2730, Y -17.0269, Z -128.0150, A 0, B 90, C 0, E1 0, E2 0, E3 0, E4 0 } C_DIS
LIN{ E6POS: X 754.1553, Y -17.0190, Z -128.0150, A 0, B 90, C 0, E1 0, E2 0, E3 0, E4 0 } C_DIS
LIN{ E6POS: X 753.1554, Y -17.0059, Z -128.0150, A 0, B 90, C 0, E1 0, E2 0, E3 0, E4 0 } C_DIS
LIN{ E6POS: X 753.0051, Y -17.0040, Z -128.0150, A 0, B 90, C 0, E1 0, E2 0, E3 0, E4 0 } C_DIS
LIN{ E6POS: X 752.0053, Y -16.9877, Z -128.0150, A 0, B 90, C 0, E1 0, E2 0, E3 0, E4 0 } C_DIS
LIN{ E6POS: X 751.0054, Y -16.9715, Z -128.0150, A 0, B 90, C 0, E1 0, E2 0, E3 0, E4 0 } C_DIS
LIN{ E6POS: X 750.0055, Y -16.9552, Z -128.0150, A 0, B 90, C 0, E1 0, E2 0, E3 0, E4 0 } C_DIS
LIN{ E6POS: X 749.0057, Y -16.9390, Z -128.0150, A 0, B 90, C 0, E1 0, E2 0, E3 0, E4 0 } C_DIS
LIN{ E6POS: X 748.0058, Y -16.9227, Z -128.0150, A 0, B 90, C 0, E1 0, E2 0, E3 0, E4 0 } C_DIS
LIN{ E6POS: X 747.0059, Y -16.9065, Z -128.0150, A 0, B 90, C 0, E1 0, E2 0, E3 0, E4 0 } C_DIS
LIN{ E6POS: X 746.3792, Y -16.8963, Z -128.0150, A 0, B 90, C 0, E1 0, E2 0, E3 0, E4 0 } C_DIS
LIN{ E6POS: X 745.4575, Y -16.9488, Z -128.0150, A 0, B 90, C 0, E1 0, E2 0, E3 0, E4 0 } C_DIS
LIN{ E6POS: X 744.4585, Y -16.9936, Z -128.0150, A 0, B 90, C 0, E1 0, E2 0, E3 0, E4 0 } C_DIS
LIN{ E6POS: X 743.4595, Y -17.0383, Z -128.0150, A 0, B 90, C 0, E1 0, E2 0, E3 0, E4 0 } C_DIS
LIN{ E6POS: X 742.4605, Y -17.0831, Z -128.0150, A 0, B 90, C 0, E1 0, E2 0, E3 0, E4 0 } C_DIS
LIN{ E6POS: X 741.4615, Y -17.1279, Z -128.0150, A 0, B 90, C 0, E1 0, E2 0, E3 0, E4 0 } C_DIS
LIN{ E6POS: X 740.4625, Y -17.1726, Z -128.0150, A 0, B 90, C 0, E1 0, E2 0, E3 0, E4 0 } C_DIS
LIN{ E6POS: X 740.1320, Y -17.1874, Z -128.0150, A 0, B 90, C 0, E1 0, E2 0, E3 0, E4 0 } C_DIS
LIN{ E6POS: X 739.5768, Y -17.3034, Z -128.0150, A 0, B 90, C 0, E1 0, E2 0, E3 0, E4 0 } C_DIS
LIN{ E6POS: X 738.5919, Y -17.4766, Z -128.0150, A 0, B 90, C 0, E1 0, E2 0, E3 0, E4 0 } C_DIS
LIN{ E6POS: X 737.6070, Y -17.6498, Z -128.0150, A 0, B 90, C 0, E1 0, E2 0, E3 0, E4 0 } C_DIS
LIN{ E6POS: X 736.6221, Y -17.8231, Z -128.0150, A 0, B 90, C 0, E1 0, E2 0, E3 0, E4 0 } C_DIS
LIN{ E6POS: X 736.3745, Y -17.8666, Z -128.0150, A 0, B 90, C 0, E1 0, E2 0, E3 0, E4 0 } C_DIS
LIN{ E6POS: X 736.1866, Y -18.0403, Z -128.0150, A 0, B 90, C 0, E1 0, E2 0, E3 0, E4 0 } C_DIS
LIN{ E6POS: X 735.4082, Y -18.6680, Z -128.0150, A 0, B 90, C 0, E1 0, E2 0, E3 0, E4 0 } C_DIS
LIN{ E6POS: X 735.1104, Y -18.9081, Z -128.0150, A 0, B 90, C 0, E1 0, E2 0, E3 0, E4 0 } C_DIS
LIN{ E6POS: X 735.7832, Y -19.6480, Z -128.0150, A 0, B 90, C 0, E1 0, E2 0, E3 0, E4 0 } C_DIS
LIN{ E6POS: X 736.1620, Y -20.0645, Z -128.0150, A 0, B 90, C 0, E1 0, E2 0, E3 0, E4 0 } C_DIS
LIN{ E6POS: X 736.3423, Y -20.2905, Z -128.0150, A 0, B 90, C 0, E1 0, E2 0, E3 0, E4 0 } C_DIS
LIN{ E6POS: X 737.2548, Y -20.6996, Z -128.0150, A 0, B 90, C 0, E1 0, E2 0, E3 0, E4 0 } C_DIS
LIN{ E6POS: X 738.1673, Y -21.1087, Z -128.0150, A 0, B 90, C 0, E1 0, E2 0, E3 0, E4 0 } C_DIS
LIN{ E6POS: X 739.0797, Y -21.5179, Z -128.0150, A 0, B 90, C 0, E1 0, E2 0, E3 0, E4 0 } C_DIS
LIN{ E6POS: X 739.5226, Y -21.7165, Z -128.0150, A 0, B 90, C 0, E1 0, E2 0, E3 0, E4 0 } C_DIS
LIN{ E6POS: X 740.0716, Y -21.9891, Z -128.0150, A 0, B 90, C 0, E1 0, E2 0, E3 0, E4 0 } C_DIS
LIN{ E6POS: X 741.0252, Y -22.2902, Z -128.0150, A 0, B 90, C 0, E1 0, E2 0, E3 0, E4 0 } C_DIS
LIN{ E6POS: X 741.9788, Y -22.5913, Z -128.0150, A 0, B 90, C 0, E1 0, E2 0, E3 0, E4 0 } C_DIS
LIN{ E6POS: X 742.9324, Y -22.8924, Z -128.0150, A 0, B 90, C 0, E1 0, E2 0, E3 0, E4 0 } C_DIS
LIN{ E6POS: X 743.8860, Y -23.1935, Z -128.0150, A 0, B 90, C 0, E1 0, E2 0, E3 0, E4 0 } C_DIS
LIN{ E6POS: X 744.8396, Y -23.4946, Z -128.0150, A 0, B 90, C 0, E1 0, E2 0, E3 0, E4 0 } C_DIS
LIN{ E6POS: X 745.3831, Y -23.6662, Z -128.0150, A 0, B 90, C 0, E1 0, E2 0, E3 0, E4 0 } C_DIS
LIN{ E6POS: X 746.3019, Y -23.9800, Z -128.0150, A 0, B 90, C 0, E1 0, E2 0, E3 0, E4 0 } C_DIS
LIN{ E6POS: X 747.2712, Y -24.2258, Z -128.0150, A 0, B 90, C 0, E1 0, E2 0, E3 0, E4 0 } C_DIS
LIN{ E6POS: X 748.2405, Y -24.4715, Z -128.0150, A 0, B 90, C 0, E1 0, E2 0, E3 0, E4 0 } C_DIS
LIN{ E6POS: X 749.2099, Y -24.7173, Z -128.0150, A 0, B 90, C 0, E1 0, E2 0, E3 0, E4 0 } C_DIS
LIN{ E6POS: X 750.1792, Y -24.9631, Z -128.0150, A 0, B 90, C 0, E1 0, E2 0, E3 0, E4 0 } C_DIS
LIN{ E6POS: X 751.1485, Y -25.2088, Z -128.0150, A 0, B 90, C 0, E1 0, E2 0, E3 0, E4 0 } C_DIS
LIN{ E6POS: X 752.1179, Y -25.4546, Z -128.0150, A 0, B 90, C 0, E1 0, E2 0, E3 0, E4 0 } C_DIS
LIN{ E6POS: X 752.9210, Y -25.6582, Z -128.0150, A 0, B 90, C 0, E1 0, E2 0, E3 0, E4 0 } C_DIS
LIN{ E6POS: X 753.8865, Y -25.9185, Z -128.0150, A 0, B 90, C 0, E1 0, E2 0, E3 0, E4 0 } C_DIS
LIN{ E6POS: X 754.0706, Y -25.9681, Z -128.0150, A 0, B 90, C 0, E1 0, E2 0, E3 0, E4 0 } C_DIS
LIN{ E6POS: X 755.0510, Y -26.1653, Z -128.0150, A 0, B 90, C 0, E1 0, E2 0, E3 0, E4 0 } C_DIS
LIN{ E6POS: X 756.0314, Y -26.3625, Z -128.0150, A 0, B 90, C 0, E1 0, E2 0, E3 0, E4 0 } C_DIS
LIN{ E6POS: X 757.0117, Y -26.5597, Z -128.0150, A 0, B 90, C 0, E1 0, E2 0, E3 0, E4 0 } C_DIS
LIN{ E6POS: X 757.9921, Y -26.7569, Z -128.0150, A 0, B 90, C 0, E1 0, E2 0, E3 0, E4 0 } C_DIS
LIN{ E6POS: X 758.9724, Y -26.9541, Z -128.0150, A 0, B 90, C 0, E1 0, E2 0, E3 0, E4 0 } C_DIS
LIN{ E6POS: X 759.9528, Y -27.1513, Z -128.0150, A 0, B 90, C 0, E1 0, E2 0, E3 0, E4 0 } C_DIS
LIN{ E6POS: X 760.9332, Y -27.3485, Z -128.0150, A 0, B 90, C 0, E1 0, E2 0, E3 0, E4 0 } C_DIS
LIN{ E6POS: X 761.1718, Y -27.3965, Z -128.0150, A 0, B 90, C 0, E1 0, E2 0, E3 0, E4 0 } C_DIS
LIN{ E6POS: X 762.1504, Y -27.6022, Z -128.0150, A 0, B 90, C 0, E1 0, E2 0, E3 0, E4 0 } C_DIS
LIN{ E6POS: X 762.4137, Y -27.6575, Z -128.0150, A 0, B 90, C 0, E1 0, E2 0, E3 0, E4 0 } C_DIS
LIN{ E6POS: X 763.4044, Y -27.7935, Z -128.0150, A 0, B 90, C 0, E1 0, E2 0, E3 0, E4 0 } C_DIS
LIN{ E6POS: X 764.3951, Y -27.9295, Z -128.0150, A 0, B 90, C 0, E1 0, E2 0, E3 0, E4 0 } C_DIS
LIN{ E6POS: X 765.3858, Y -28.0655, Z -128.0150, A 0, B 90, C 0, E1 0, E2 0, E3 0, E4 0 } C_DIS
LIN{ E6POS: X 766.3766, Y -28.2014, Z -128.0150, A 0, B 90, C 0, E1 0, E2 0, E3 0, E4 0 } C_DIS
LIN{ E6POS: X 767.3673, Y -28.3374, Z -128.0150, A 0, B 90, C 0, E1 0, E2 0, E3 0, E4 0 } C_DIS
LIN{ E6POS: X 768.3580, Y -28.4734, Z -128.0150, A 0, B 90, C 0, E1 0, E2 0, E3 0, E4 0 } C_DIS
LIN{ E6POS: X 769.1744, Y -28.5854, Z -128.0150, A 0, B 90, C 0, E1 0, E2 0, E3 0, E4 0 } C_DIS
LIN{ E6POS: X 770.1648, Y -28.7238, Z -128.0150, A 0, B 90, C 0, E1 0, E2 0, E3 0, E4 0 } C_DIS
LIN{ E6POS: X 770.3698, Y -28.7524, Z -128.0150, A 0, B 90, C 0, E1 0, E2 0, E3 0, E4 0 } C_DIS
LIN{ E6POS: X 771.3693, Y -28.7841, Z -128.0150, A 0, B 90, C 0, E1 0, E2 0, E3 0, E4 0 } C_DIS
LIN{ E6POS: X 772.3688, Y -28.8158, Z -128.0150, A 0, B 90, C 0, E1 0, E2 0, E3 0, E4 0 } C_DIS
LIN{ E6POS: X 773.3683, Y -28.8475, Z -128.0150, A 0, B 90, C 0, E1 0, E2 0, E3 0, E4 0 } C_DIS
LIN{ E6POS: X 774.3678, Y -28.8792, Z -128.0150, A 0, B 90, C 0, E1 0, E2 0, E3 0, E4 0 } C_DIS
LIN{ E6POS: X 775.3673, Y -28.9109, Z -128.0150, A 0, B 90, C 0, E1 0, E2 0, E3 0, E4 0 } C_DIS
LIN{ E6POS: X 775.9642, Y -28.9298, Z -128.0150, A 0, B 90, C 0, E1 0, E2 0, E3 0, E4 0 } C_DIS
LIN{ E6POS: X 776.9638, Y -28.9573, Z -128.0150, A 0, B 90, C 0, E1 0, E2 0, E3 0, E4 0 } C_DIS
LIN{ E6POS: X 776.9745, Y -28.9576, Z -128.0150, A 0, B 90, C 0, E1 0, E2 0, E3 0, E4 0 } C_DIS
LIN{ E6POS: X 777.9572, Y -29.1432, Z -128.0150, A 0, B 90, C 0, E1 0, E2 0, E3 0, E4 0 } C_DIS
LIN{ E6POS: X 778.9398, Y -29.3289, Z -128.0150, A 0, B 90, C 0, E1 0, E2 0, E3 0, E4 0 } C_DIS
LIN{ E6POS: X 779.9224, Y -29.5145, Z -128.0150, A 0, B 90, C 0, E1 0, E2 0, E3 0, E4 0 } C_DIS
LIN{ E6POS: X 780.9050, Y -29.7001, Z -128.0150, A 0, B 90, C 0, E1 0, E2 0, E3 0, E4 0 } C_DIS
LIN{ E6POS: X 781.2002, Y -29.7558, Z -128.0150, A 0, B 90, C 0, E1 0, E2 0, E3 0, E4 0 } C_DIS
LIN{ E6POS: X 781.9775, Y -29.9049, Z -128.0150, A 0, B 90, C 0, E1 0, E2 0, E3 0, E4 0 } C_DIS
LIN{ E6POS: X 782.6666, Y -30.6295, Z -128.0150, A 0, B 90, C 0, E1 0, E2 0, E3 0, E4 0 } C_DIS
LIN{ E6POS: X 783.3558, Y -31.3541, Z -128.0150, A 0, B 90, C 0, E1 0, E2 0, E3 0, E4 0 } C_DIS
LIN{ E6POS: X 784.0449, Y -32.0788, Z -128.0150, A 0, B 90, C 0, E1 0, E2 0, E3 0, E4 0 } C_DIS
LIN{ E6POS: X 784.6318, Y -32.6959, Z -128.0150, A 0, B 90, C 0, E1 0, E2 0, E3 0, E4 0 } C_DIS
LIN{ E6POS: X 785.1281, Y -33.2266, Z -128.0150, A 0, B 90, C 0, E1 0, E2 0, E3 0, E4 0 } C_DIS
LIN{ E6POS: X 785.2695, Y -34.2166, Z -128.0150, A 0, B 90, C 0, E1 0, E2 0, E3 0, E4 0 } C_DIS
LIN{ E6POS: X 785.4109, Y -35.2065, Z -128.0150, A 0, B 90, C 0, E1 0, E2 0, E3 0, E4 0 } C_DIS
LIN{ E6POS: X 785.5523, Y -36.1965, Z -128.0150, A 0, B 90, C 0, E1 0, E2 0, E3 0, E4 0 } C_DIS
LIN{ E6POS: X 785.6937, Y -37.1864, Z -128.0150, A 0, B 90, C 0, E1 0, E2 0, E3 0, E4 0 } C_DIS
LIN{ E6POS: X 785.8351, Y -38.1764, Z -128.0150, A 0, B 90, C 0, E1 0, E2 0, E3 0, E4 0 } C_DIS
LIN{ E6POS: X 785.9765, Y -39.1663, Z -128.0150, A 0, B 90, C 0, E1 0, E2 0, E3 0, E4 0 } C_DIS
LIN{ E6POS: X 786.0072, Y -39.3813, Z -128.0150, A 0, B 90, C 0, E1 0, E2 0, E3 0, E4 0 } C_DIS
LIN{ E6POS: X 786.1486, Y -40.3712, Z -128.0150, A 0, B 90, C 0, E1 0, E2 0, E3 0, E4 0 } C_DIS
LIN{ E6POS: X 786.1747, Y -40.5536, Z -128.0150, A 0, B 90, C 0, E1 0, E2 0, E3 0, E4 0 } C_DIS
LIN{ E6POS: X 786.0743, Y -41.5485, Z -128.0150, A 0, B 90, C 0, E1 0, E2 0, E3 0, E4 0 } C_DIS
LIN{ E6POS: X 785.9740, Y -42.5435, Z -128.0150, A 0, B 90, C 0, E1 0, E2 0, E3 0, E4 0 } C_DIS
LIN{ E6POS: X 785.8737, Y -43.5384, Z -128.0150, A 0, B 90, C 0, E1 0, E2 0, E3 0, E4 0 } C_DIS
LIN{ E6POS: X 785.7734, Y -44.5334, Z -128.0150, A 0, B 90, C 0, E1 0, E2 0, E3 0, E4 0 } C_DIS
LIN{ E6POS: X 785.6731, Y -45.5283, Z -128.0150, A 0, B 90, C 0, E1 0, E2 0, E3 0, E4 0 } C_DIS
LIN{ E6POS: X 785.5728, Y -46.5233, Z -128.0150, A 0, B 90, C 0, E1 0, E2 0, E3 0, E4 0 } C_DIS
LIN{ E6POS: X 785.4725, Y -47.5183, Z -128.0150, A 0, B 90, C 0, E1 0, E2 0, E3 0, E4 0 } C_DIS
LIN{ E6POS: X 785.3721, Y -48.5132, Z -128.0150, A 0, B 90, C 0, E1 0, E2 0, E3 0, E4 0 } C_DIS
LIN{ E6POS: X 785.2718, Y -49.5082, Z -128.0150, A 0, B 90, C 0, E1 0, E2 0, E3 0, E4 0 } C_DIS
LIN{ E6POS: X 785.1715, Y -50.5031, Z -128.0150, A 0, B 90, C 0, E1 0, E2 0, E3 0, E4 0 } C_DIS
LIN{ E6POS: X 785.0766, Y -51.4441, Z -128.0150, A 0, B 90, C 0, E1 0, E2 0, E3 0, E4 0 } C_DIS
LIN{ E6POS: X 784.9763, Y -52.4390, Z -128.0150, A 0, B 90, C 0, E1 0, E2 0, E3 0, E4 0 } C_DIS
LIN{ E6POS: X 784.8760, Y -53.4340, Z -128.0150, A 0, B 90, C 0, E1 0, E2 0, E3 0, E4 0 } C_DIS
LIN{ E6POS: X 784.8675, Y -53.5185, Z -128.0150, A 0, B 90, C 0, E1 0, E2 0, E3 0, E4 0 } C_DIS
LIN{ E6POS: X 784.6915, Y -54.5029, Z -128.0150, A 0, B 90, C 0, E1 0, E2 0, E3 0, E4 0 } C_DIS
LIN{ E6POS: X 784.5156, Y -55.4873, Z -128.0150, A 0, B 90, C 0, E1 0, E2 0, E3 0, E4 0 } C_DIS
LIN{ E6POS: X 784.3396, Y -56.4717, Z -128.0150, A 0, B 90, C 0, E1 0, E2 0, E3 0, E4 0 } C_DIS
LIN{ E6POS: X 784.1637, Y -57.4560, Z -128.0150, A 0, B 90, C 0, E1 0, E2 0, E3 0, E4 0 } C_DIS
LIN{ E6POS: X 783.9877, Y -58.4404, Z -128.0150, A 0, B 90, C 0, E1 0, E2 0, E3 0, E4 0 } C_DIS
LIN{ E6POS: X 783.8118, Y -59.4248, Z -128.0150, A 0, B 90, C 0, E1 0, E2 0, E3 0, E4 0 } C_DIS
LIN{ E6POS: X 783.6358, Y -60.4092, Z -128.0150, A 0, B 90, C 0, E1 0, E2 0, E3 0, E4 0 } C_DIS
LIN{ E6POS: X 783.4599, Y -61.3936, Z -128.0150, A 0, B 90, C 0, E1 0, E2 0, E3 0, E4 0 } C_DIS
LIN{ E6POS: X 783.2839, Y -62.3780, Z -128.0150, A 0, B 90, C 0, E1 0, E2 0, E3 0, E4 0 } C_DIS
LIN{ E6POS: X 783.1080, Y -63.3624, Z -128.0150, A 0, B 90, C 0, E1 0, E2 0, E3 0, E4 0 } C_DIS
LIN{ E6POS: X 782.9320, Y -64.3468, Z -128.0150, A 0, B 90, C 0, E1 0, E2 0, E3 0, E4 0 } C_DIS
LIN{ E6POS: X 782.7561, Y -65.3312, Z -128.0150, A 0, B 90, C 0, E1 0, E2 0, E3 0, E4 0 } C_DIS
LIN{ E6POS: X 782.5801, Y -66.3156, Z -128.0150, A 0, B 90, C 0, E1 0, E2 0, E3 0, E4 0 } C_DIS
LIN{ E6POS: X 782.4042, Y -67.3000, Z -128.0150, A 0, B 90, C 0, E1 0, E2 0, E3 0, E4 0 } C_DIS
LIN{ E6POS: X 782.2861, Y -67.9609, Z -128.0150, A 0, B 90, C 0, E1 0, E2 0, E3 0, E4 0 } C_DIS
LIN{ E6POS: X 782.1101, Y -68.9453, Z -128.0150, A 0, B 90, C 0, E1 0, E2 0, E3 0, E4 0 } C_DIS
LIN{ E6POS: X 781.9341, Y -69.9297, Z -128.0150, A 0, B 90, C 0, E1 0, E2 0, E3 0, E4 0 } C_DIS
LIN{ E6POS: X 781.7943, Y -70.7119, Z -128.0150, A 0, B 90, C 0, E1 0, E2 0, E3 0, E4 0 } C_DIS
LIN{ E6POS: X 781.5865, Y -71.6900, Z -128.0150, A 0, B 90, C 0, E1 0, E2 0, E3 0, E4 0 } C_DIS
LIN{ E6POS: X 781.3787, Y -72.6682, Z -128.0150, A 0, B 90, C 0, E1 0, E2 0, E3 0, E4 0 } C_DIS
LIN{ E6POS: X 781.1709, Y -73.6464, Z -128.0150, A 0, B 90, C 0, E1 0, E2 0, E3 0, E4 0 } C_DIS
LIN{ E6POS: X 780.9631, Y -74.6245, Z -128.0150, A 0, B 90, C 0, E1 0, E2 0, E3 0, E4 0 } C_DIS
LIN{ E6POS: X 780.7553, Y -75.6027, Z -128.0150, A 0, B 90, C 0, E1 0, E2 0, E3 0, E4 0 } C_DIS
LIN{ E6POS: X 780.5475, Y -76.5809, Z -128.0150, A 0, B 90, C 0, E1 0, E2 0, E3 0, E4 0 } C_DIS
LIN{ E6POS: X 780.3397, Y -77.5590, Z -128.0150, A 0, B 90, C 0, E1 0, E2 0, E3 0, E4 0 } C_DIS
LIN{ E6POS: X 780.1319, Y -78.5372, Z -128.0150, A 0, B 90, C 0, E1 0, E2 0, E3 0, E4 0 } C_DIS
LIN{ E6POS: X 779.9241, Y -79.5154, Z -128.0150, A 0, B 90, C 0, E1 0, E2 0, E3 0, E4 0 } C_DIS
LIN{ E6POS: X 779.7163, Y -80.4936, Z -128.0150, A 0, B 90, C 0, E1 0, E2 0, E3 0, E4 0 } C_DIS
LIN{ E6POS: X 779.5085, Y -81.4717, Z -128.0150, A 0, B 90, C 0, E1 0, E2 0, E3 0, E4 0 } C_DIS
LIN{ E6POS: X 779.3007, Y -82.4499, Z -128.0150, A 0, B 90, C 0, E1 0, E2 0, E3 0, E4 0 } C_DIS
LIN{ E6POS: X 779.0929, Y -83.4281, Z -128.0150, A 0, B 90, C 0, E1 0, E2 0, E3 0, E4 0 } C_DIS
LIN{ E6POS: X 778.8851, Y -84.4062, Z -128.0150, A 0, B 90, C 0, E1 0, E2 0, E3 0, E4 0 } C_DIS
LIN{ E6POS: X 778.6773, Y -85.3844, Z -128.0150, A 0, B 90, C 0, E1 0, E2 0, E3 0, E4 0 } C_DIS
LIN{ E6POS: X 778.4695, Y -86.3626, Z -128.0150, A 0, B 90, C 0, E1 0, E2 0, E3 0, E4 0 } C_DIS
LIN{ E6POS: X 778.2617, Y -87.3408, Z -128.0150, A 0, B 90, C 0, E1 0, E2 0, E3 0, E4 0 } C_DIS
LIN{ E6POS: X 778.2231, Y -87.5223, Z -128.0150, A 0, B 90, C 0, E1 0, E2 0, E3 0, E4 0 } C_DIS
LIN{ E6POS: X 778.0153, Y -88.5005, Z -128.0150, A 0, B 90, C 0, E1 0, E2 0, E3 0, E4 0 } C_DIS
LIN{ E6POS: X 777.8075, Y -89.4786, Z -128.0150, A 0, B 90, C 0, E1 0, E2 0, E3 0, E4 0 } C_DIS
LIN{ E6POS: X 777.5997, Y -90.4568, Z -128.0150, A 0, B 90, C 0, E1 0, E2 0, E3 0, E4 0 } C_DIS
LIN{ E6POS: X 777.5429, Y -90.7243, Z -128.0150, A 0, B 90, C 0, E1 0, E2 0, E3 0, E4 0 } C_DIS
LIN{ E6POS: X 777.3226, Y -91.6997, Z -128.0150, A 0, B 90, C 0, E1 0, E2 0, E3 0, E4 0 } C_DIS
LIN{ E6POS: X 777.1022, Y -92.6751, Z -128.0150, A 0, B 90, C 0, E1 0, E2 0, E3 0, E4 0 } C_DIS
LIN{ E6POS: X 776.8819, Y -93.6506, Z -128.0150, A 0, B 90, C 0, E1 0, E2 0, E3 0, E4 0 } C_DIS
LIN{ E6POS: X 776.6615, Y -94.6260, Z -128.0150, A 0, B 90, C 0, E1 0, E2 0, E3 0, E4 0 } C_DIS
LIN{ E6POS: X 776.4412, Y -95.6014, Z -128.0150, A 0, B 90, C 0, E1 0, E2 0, E3 0, E4 0 } C_DIS
LIN{ E6POS: X 776.2208, Y -96.5768, Z -128.0150, A 0, B 90, C 0, E1 0, E2 0, E3 0, E4 0 } C_DIS
LIN{ E6POS: X 776.0005, Y -97.5522, Z -128.0150, A 0, B 90, C 0, E1 0, E2 0, E3 0, E4 0 } C_DIS
LIN{ E6POS: X 775.7802, Y -98.5277, Z -128.0150, A 0, B 90, C 0, E1 0, E2 0, E3 0, E4 0 } C_DIS
LIN{ E6POS: X 775.5598, Y -99.5031, Z -128.0150, A 0, B 90, C 0, E1 0, E2 0, E3 0, E4 0 } C_DIS
LIN{ E6POS: X 775.3395, Y -100.4785, Z -128.0150, A 0, B 90, C 0, E1 0, E2 0, E3 0, E4 0 } C_DIS
LIN{ E6POS: X 775.1191, Y -101.4539, Z -128.0150, A 0, B 90, C 0, E1 0, E2 0, E3 0, E4 0 } C_DIS
LIN{ E6POS: X 774.8988, Y -102.4294, Z -128.0150, A 0, B 90, C 0, E1 0, E2 0, E3 0, E4 0 } C_DIS
LIN{ E6POS: X 774.6784, Y -103.4048, Z -128.0150, A 0, B 90, C 0, E1 0, E2 0, E3 0, E4 0 } C_DIS
LIN{ E6POS: X 774.4581, Y -104.3802, Z -128.0150, A 0, B 90, C 0, E1 0, E2 0, E3 0, E4 0 } C_DIS
LIN{ E6POS: X 774.2377, Y -105.3556, Z -128.0150, A 0, B 90, C 0, E1 0, E2 0, E3 0, E4 0 } C_DIS
LIN{ E6POS: X 774.0174, Y -106.3310, Z -128.0150, A 0, B 90, C 0, E1 0, E2 0, E3 0, E4 0 } C_DIS
LIN{ E6POS: X 773.7970, Y -107.3065, Z -128.0150, A 0, B 90, C 0, E1 0, E2 0, E3 0, E4 0 } C_DIS
LIN{ E6POS: X 773.5767, Y -108.2819, Z -128.0150, A 0, B 90, C 0, E1 0, E2 0, E3 0, E4 0 } C_DIS
LIN{ E6POS: X 773.4780, Y -108.7187, Z -128.0150, A 0, B 90, C 0, E1 0, E2 0, E3 0, E4 0 } C_DIS
LIN{ E6POS: X 773.2577, Y -109.6941, Z -128.0150, A 0, B 90, C 0, E1 0, E2 0, E3 0, E4 0 } C_DIS
LIN{ E6POS: X 773.0373, Y -110.6695, Z -128.0150, A 0, B 90, C 0, E1 0, E2 0, E3 0, E4 0 } C_DIS
LIN{ E6POS: X 772.8170, Y -111.6450, Z -128.0150, A 0, B 90, C 0, E1 0, E2 0, E3 0, E4 0 } C_DIS
LIN{ E6POS: X 772.7038, Y -112.1462, Z -128.0150, A 0, B 90, C 0, E1 0, E2 0, E3 0, E4 0 } C_DIS
LIN{ E6POS: X 772.0412, Y -111.3972, Z -128.0150, A 0, B 90, C 0, E1 0, E2 0, E3 0, E4 0 } C_DIS
LIN{ E6POS: X 771.3787, Y -110.6481, Z -128.0150, A 0, B 90, C 0, E1 0, E2 0, E3 0, E4 0 } C_DIS
LIN{ E6POS: X 770.7162, Y -109.8991, Z -128.0150, A 0, B 90, C 0, E1 0, E2 0, E3 0, E4 0 } C_DIS
LIN{ E6POS: X 770.4591, Y -109.6084, Z -128.0150, A 0, B 90, C 0, E1 0, E2 0, E3 0, E4 0 } C_DIS
LIN{ E6POS: X 770.0315, Y -109.1250, Z -128.0150, A 0, B 90, C 0, E1 0, E2 0, E3 0, E4 0 } C_DIS
LIN{ E6POS: X 769.2905, Y -108.4535, Z -128.0150, A 0, B 90, C 0, E1 0, E2 0, E3 0, E4 0 } C_DIS
LIN{ E6POS: X 768.5495, Y -107.7819, Z -128.0150, A 0, B 90, C 0, E1 0, E2 0, E3 0, E4 0 } C_DIS
LIN{ E6POS: X 767.8086, Y -107.1104, Z -128.0150, A 0, B 90, C 0, E1 0, E2 0, E3 0, E4 0 } C_DIS
LIN{ E6POS: X 767.1113, Y -106.4786, Z -128.0150, A 0, B 90, C 0, E1 0, E2 0, E3 0, E4 0 } C_DIS
LIN{ E6POS: X 766.5590, Y -105.9769, Z -128.0150, A 0, B 90, C 0, E1 0, E2 0, E3 0, E4 0 } C_DIS
LIN{ E6POS: X 765.7575, Y -105.4385, Z -128.0150, A 0, B 90, C 0, E1 0, E2 0, E3 0, E4 0 } C_DIS
LIN{ E6POS: X 764.9268, Y -104.8818, Z -128.0150, A 0, B 90, C 0, E1 0, E2 0, E3 0, E4 0 } C_DIS
LIN{ E6POS: X 764.0961, Y -104.3251, Z -128.0150, A 0, B 90, C 0, E1 0, E2 0, E3 0, E4 0 } C_DIS
LIN{ E6POS: X 763.2654, Y -103.7683, Z -128.0150, A 0, B 90, C 0, E1 0, E2 0, E3 0, E4 0 } C_DIS
LIN{ E6POS: X 762.4347, Y -103.2116, Z -128.0150, A 0, B 90, C 0, E1 0, E2 0, E3 0, E4 0 } C_DIS
LIN{ E6POS: X 761.6040, Y -102.6549, Z -128.0150, A 0, B 90, C 0, E1 0, E2 0, E3 0, E4 0 } C_DIS
LIN{ E6POS: X 761.4881, Y -102.5772, Z -128.0150, A 0, B 90, C 0, E1 0, E2 0, E3 0, E4 0 } C_DIS
LIN{ E6POS: X 760.5955, Y -102.1265, Z -128.0150, A 0, B 90, C 0, E1 0, E2 0, E3 0, E4 0 } C_DIS
LIN{ E6POS: X 760.3127, Y -101.9838, Z -128.0150, A 0, B 90, C 0, E1 0, E2 0, E3 0, E4 0 } C_DIS
LIN{ E6POS: X 759.4205, Y -101.5322, Z -128.0150, A 0, B 90, C 0, E1 0, E2 0, E3 0, E4 0 } C_DIS
LIN{ E6POS: X 758.5282, Y -101.0806, Z -128.0150, A 0, B 90, C 0, E1 0, E2 0, E3 0, E4 0 } C_DIS
LIN{ E6POS: X 757.6360, Y -100.6291, Z -128.0150, A 0, B 90, C 0, E1 0, E2 0, E3 0, E4 0 } C_DIS
LIN{ E6POS: X 756.7438, Y -100.1775, Z -128.0150, A 0, B 90, C 0, E1 0, E2 0, E3 0, E4 0 } C_DIS
LIN{ E6POS: X 755.8515, Y -99.7259, Z -128.0150, A 0, B 90, C 0, E1 0, E2 0, E3 0, E4 0 } C_DIS
LIN{ E6POS: X 754.9593, Y -99.2743, Z -128.0150, A 0, B 90, C 0, E1 0, E2 0, E3 0, E4 0 } C_DIS
LIN{ E6POS: X 754.0671, Y -98.8228, Z -128.0150, A 0, B 90, C 0, E1 0, E2 0, E3 0, E4 0 } C_DIS
LIN{ E6POS: X 754.0181, Y -98.7980, Z -128.0150, A 0, B 90, C 0, E1 0, E2 0, E3 0, E4 0 } C_DIS
LIN{ E6POS: X 753.0891, Y -98.4281, Z -128.0150, A 0, B 90, C 0, E1 0, E2 0, E3 0, E4 0 } C_DIS
LIN{ E6POS: X 752.3440, Y -98.1315, Z -128.0150, A 0, B 90, C 0, E1 0, E2 0, E3 0, E4 0 } C_DIS
LIN{ E6POS: X 751.4162, Y -97.7582, Z -128.0150, A 0, B 90, C 0, E1 0, E2 0, E3 0, E4 0 } C_DIS
LIN{ E6POS: X 750.4885, Y -97.3850, Z -128.0150, A 0, B 90, C 0, E1 0, E2 0, E3 0, E4 0 } C_DIS
LIN{ E6POS: X 749.5608, Y -97.0117, Z -128.0150, A 0, B 90, C 0, E1 0, E2 0, E3 0, E4 0 } C_DIS
LIN{ E6POS: X 748.6330, Y -96.6385, Z -128.0150, A 0, B 90, C 0, E1 0, E2 0, E3 0, E4 0 } C_DIS
LIN{ E6POS: X 747.7053, Y -96.2652, Z -128.0150, A 0, B 90, C 0, E1 0, E2 0, E3 0, E4 0 } C_DIS
LIN{ E6POS: X 746.7776, Y -95.8920, Z -128.0150, A 0, B 90, C 0, E1 0, E2 0, E3 0, E4 0 } C_DIS
LIN{ E6POS: X 745.8498, Y -95.5187, Z -128.0150, A 0, B 90, C 0, E1 0, E2 0, E3 0, E4 0 } C_DIS
LIN{ E6POS: X 744.9221, Y -95.1455, Z -128.0150, A 0, B 90, C 0, E1 0, E2 0, E3 0, E4 0 } C_DIS
LIN{ E6POS: X 743.9944, Y -94.7722, Z -128.0150, A 0, B 90, C 0, E1 0, E2 0, E3 0, E4 0 } C_DIS
LIN{ E6POS: X 743.3502, Y -94.5130, Z -128.0150, A 0, B 90, C 0, E1 0, E2 0, E3 0, E4 0 } C_DIS
LIN{ E6POS: X 742.4085, Y -94.1765, Z -128.0150, A 0, B 90, C 0, E1 0, E2 0, E3 0, E4 0 } C_DIS
LIN{ E6POS: X 741.4669, Y -93.8399, Z -128.0150, A 0, B 90, C 0, E1 0, E2 0, E3 0, E4 0 } C_DIS
LIN{ E6POS: X 741.4554, Y -93.8358, Z -128.0150, A 0, B 90, C 0, E1 0, E2 0, E3 0, E4 0 } C_DIS
LIN{ E6POS: X 740.5151, Y -93.4955, Z -128.0150, A 0, B 90, C 0, E1 0, E2 0, E3 0, E4 0 } C_DIS
LIN{ E6POS: X 739.5748, Y -93.1553, Z -128.0150, A 0, B 90, C 0, E1 0, E2 0, E3 0, E4 0 } C_DIS
LIN{ E6POS: X 738.6344, Y -92.8150, Z -128.0150, A 0, B 90, C 0, E1 0, E2 0, E3 0, E4 0 } C_DIS
LIN{ E6POS: X 737.6941, Y -92.4747, Z -128.0150, A 0, B 90, C 0, E1 0, E2 0, E3 0, E4 0 } C_DIS
LIN{ E6POS: X 736.7538, Y -92.1345, Z -128.0150, A 0, B 90, C 0, E1 0, E2 0, E3 0, E4 0 } C_DIS
LIN{ E6POS: X 735.8134, Y -91.7942, Z -128.0150, A 0, B 90, C 0, E1 0, E2 0, E3 0, E4 0 } C_DIS
LIN{ E6POS: X 734.8731, Y -91.4540, Z -128.0150, A 0, B 90, C 0, E1 0, E2 0, E3 0, E4 0 } C_DIS
LIN{ E6POS: X 733.9328, Y -91.1137, Z -128.0150, A 0, B 90, C 0, E1 0, E2 0, E3 0, E4 0 } C_DIS
LIN{ E6POS: X 732.9924, Y -90.7735, Z -128.0150, A 0, B 90, C 0, E1 0, E2 0, E3 0, E4 0 } C_DIS
LIN{ E6POS: X 732.0521, Y -90.4332, Z -128.0150, A 0, B 90, C 0, E1 0, E2 0, E3 0, E4 0 } C_DIS
LIN{ E6POS: X 731.2583, Y -90.1460, Z -128.0150, A 0, B 90, C 0, E1 0, E2 0, E3 0, E4 0 } C_DIS
LIN{ E6POS: X 730.3116, Y -89.8239, Z -128.0150, A 0, B 90, C 0, E1 0, E2 0, E3 0, E4 0 } C_DIS
LIN{ E6POS: X 729.4206, Y -89.5207, Z -128.0150, A 0, B 90, C 0, E1 0, E2 0, E3 0, E4 0 } C_DIS
LIN{ E6POS: X 728.4748, Y -89.1958, Z -128.0150, A 0, B 90, C 0, E1 0, E2 0, E3 0, E4 0 } C_DIS
LIN{ E6POS: X 727.5291, Y -88.8709, Z -128.0150, A 0, B 90, C 0, E1 0, E2 0, E3 0, E4 0 } C_DIS
LIN{ E6POS: X 726.5833, Y -88.5460, Z -128.0150, A 0, B 90, C 0, E1 0, E2 0, E3 0, E4 0 } C_DIS
LIN{ E6POS: X 725.6376, Y -88.2211, Z -128.0150, A 0, B 90, C 0, E1 0, E2 0, E3 0, E4 0 } C_DIS
LIN{ E6POS: X 724.6918, Y -87.8962, Z -128.0150, A 0, B 90, C 0, E1 0, E2 0, E3 0, E4 0 } C_DIS
LIN{ E6POS: X 723.7461, Y -87.5713, Z -128.0150, A 0, B 90, C 0, E1 0, E2 0, E3 0, E4 0 } C_DIS
LIN{ E6POS: X 722.8003, Y -87.2464, Z -128.0150, A 0, B 90, C 0, E1 0, E2 0, E3 0, E4 0 } C_DIS
LIN{ E6POS: X 721.8546, Y -86.9215, Z -128.0150, A 0, B 90, C 0, E1 0, E2 0, E3 0, E4 0 } C_DIS
LIN{ E6POS: X 720.9088, Y -86.5966, Z -128.0150, A 0, B 90, C 0, E1 0, E2 0, E3 0, E4 0 } C_DIS
LIN{ E6POS: X 719.9631, Y -86.2717, Z -128.0150, A 0, B 90, C 0, E1 0, E2 0, E3 0, E4 0 } C_DIS
LIN{ E6POS: X 719.5166, Y -86.1183, Z -128.0150, A 0, B 90, C 0, E1 0, E2 0, E3 0, E4 0 } C_DIS
LIN{ E6POS: X 718.5698, Y -85.7966, Z -128.0150, A 0, B 90, C 0, E1 0, E2 0, E3 0, E4 0 } C_DIS
LIN{ E6POS: X 718.0137, Y -85.6076, Z -128.0150, A 0, B 90, C 0, E1 0, E2 0, E3 0, E4 0 } C_DIS
LIN{ E6POS: X 717.0668, Y -85.2860, Z -128.0150, A 0, B 90, C 0, E1 0, E2 0, E3 0, E4 0 } C_DIS
LIN{ E6POS: X 716.1199, Y -84.9645, Z -128.0150, A 0, B 90, C 0, E1 0, E2 0, E3 0, E4 0 } C_DIS
LIN{ E6POS: X 715.1730, Y -84.6430, Z -128.0150, A 0, B 90, C 0, E1 0, E2 0, E3 0, E4 0 } C_DIS
LIN{ E6POS: X 714.2261, Y -84.3215, Z -128.0150, A 0, B 90, C 0, E1 0, E2 0, E3 0, E4 0 } C_DIS
LIN{ E6POS: X 713.2792, Y -83.9999, Z -128.0150, A 0, B 90, C 0, E1 0, E2 0, E3 0, E4 0 } C_DIS
LIN{ E6POS: X 712.3323, Y -83.6784, Z -128.0150, A 0, B 90, C 0, E1 0, E2 0, E3 0, E4 0 } C_DIS
LIN{ E6POS: X 711.3854, Y -83.3569, Z -128.0150, A 0, B 90, C 0, E1 0, E2 0, E3 0, E4 0 } C_DIS
LIN{ E6POS: X 710.4385, Y -83.0354, Z -128.0150, A 0, B 90, C 0, E1 0, E2 0, E3 0, E4 0 } C_DIS
LIN{ E6POS: X 709.9000, Y -82.8525, Z -128.0150, A 0, B 90, C 0, E1 0, E2 0, E3 0, E4 0 } C_DIS
LIN{ E6POS: X 709.0099, Y -82.5191, Z -128.0150, A 0, B 90, C 0, E1 0, E2 0, E3 0, E4 0 } C_DIS
LIN{ E6POS: X 708.0696, Y -82.1788, Z -128.0150, A 0, B 90, C 0, E1 0, E2 0, E3 0, E4 0 } C_DIS
LIN{ E6POS: X 707.1293, Y -81.8385, Z -128.0150, A 0, B 90, C 0, E1 0, E2 0, E3 0, E4 0 } C_DIS
LIN{ E6POS: X 706.1890, Y -81.4981, Z -128.0150, A 0, B 90, C 0, E1 0, E2 0, E3 0, E4 0 } C_DIS
LIN{ E6POS: X 705.2487, Y -81.1578, Z -128.0150, A 0, B 90, C 0, E1 0, E2 0, E3 0, E4 0 } C_DIS
LIN{ E6POS: X 704.3084, Y -80.8174, Z -128.0150, A 0, B 90, C 0, E1 0, E2 0, E3 0, E4 0 } C_DIS
LIN{ E6POS: X 704.1818, Y -80.7716, Z -128.0150, A 0, B 90, C 0, E1 0, E2 0, E3 0, E4 0 } C_DIS
LIN{ E6POS: X 703.7511, Y -80.5712, Z -128.0150, A 0, B 90, C 0, E1 0, E2 0, E3 0, E4 0 } C_DIS
LIN{ E6POS: X 702.8290, Y -80.1842, Z -128.0150, A 0, B 90, C 0, E1 0, E2 0, E3 0, E4 0 } C_DIS
LIN{ E6POS: X 701.9069, Y -79.7972, Z -128.0150, A 0, B 90, C 0, E1 0, E2 0, E3 0, E4 0 } C_DIS
LIN{ E6POS: X 701.3873, Y -79.5791, Z -128.0150, A 0, B 90, C 0, E1 0, E2 0, E3 0, E4 0 } C_DIS
LIN{ E6POS: X 701.2824, Y -79.4222, Z -128.0150, A 0, B 90, C 0, E1 0, E2 0, E3 0, E4 0 } C_DIS
LIN{ E6POS: X 700.6304, Y -78.7761, Z -128.0150, A 0, B 90, C 0, E1 0, E2 0, E3 0, E4 0 } C_DIS
LIN{ E6POS: X 700.8681, Y -77.8047, Z -128.0150, A 0, B 90, C 0, E1 0, E2 0, E3 0, E4 0 } C_DIS
LIN{ E6POS: X 700.9392, Y -77.5141, Z -128.0150, A 0, B 90, C 0, E1 0, E2 0, E3 0, E4 0 } C_DIS
LIN{ E6POS: X 701.0124, Y -77.2533, Z -128.0150, A 0, B 90, C 0, E1 0, E2 0, E3 0, E4 0 } C_DIS
LIN{ E6POS: X 701.2425, Y -76.2801, Z -128.0150, A 0, B 90, C 0, E1 0, E2 0, E3 0, E4 0 } C_DIS
LIN{ E6POS: X 701.2917, Y -76.0721, Z -128.0150, A 0, B 90, C 0, E1 0, E2 0, E3 0, E4 0 } C_DIS
LIN{ E6POS: X 701.3553, Y -75.8362, Z -128.0150, A 0, B 90, C 0, E1 0, E2 0, E3 0, E4 0 } C_DIS
LIN{ E6POS: X 701.5909, Y -74.8643, Z -128.0150, A 0, B 90, C 0, E1 0, E2 0, E3 0, E4 0 } C_DIS
LIN{ E6POS: X 701.6406, Y -74.6594, Z -128.0150, A 0, B 90, C 0, E1 0, E2 0, E3 0, E4 0 } C_DIS
LIN{ E6POS: X 701.7043, Y -74.4279, Z -128.0150, A 0, B 90, C 0, E1 0, E2 0, E3 0, E4 0 } C_DIS
LIN{ E6POS: X 701.9492, Y -73.4584, Z -128.0150, A 0, B 90, C 0, E1 0, E2 0, E3 0, E4 0 } C_DIS
LIN{ E6POS: X 701.9996, Y -73.2587, Z -128.0150, A 0, B 90, C 0, E1 0, E2 0, E3 0, E4 0 } C_DIS
LIN{ E6POS: X 702.0637, Y -73.0341, Z -128.0150, A 0, B 90, C 0, E1 0, E2 0, E3 0, E4 0 } C_DIS
LIN{ E6POS: X 702.3196, Y -72.0674, Z -128.0150, A 0, B 90, C 0, E1 0, E2 0, E3 0, E4 0 } C_DIS
LIN{ E6POS: X 702.3713, Y -71.8722, Z -128.0150, A 0, B 90, C 0, E1 0, E2 0, E3 0, E4 0 } C_DIS
LIN{ E6POS: X 702.4358, Y -71.6567, Z -128.0150, A 0, B 90, C 0, E1 0, E2 0, E3 0, E4 0 } C_DIS
LIN{ E6POS: X 702.6960, Y -70.6911, Z -128.0150, A 0, B 90, C 0, E1 0, E2 0, E3 0, E4 0 } C_DIS
LIN{ E6POS: X 702.7500, Y -70.4908, Z -128.0150, A 0, B 90, C 0, E1 0, E2 0, E3 0, E4 0 } C_DIS
LIN{ E6POS: X 702.8141, Y -70.2790, Z -128.0150, A 0, B 90, C 0, E1 0, E2 0, E3 0, E4 0 } C_DIS
LIN{ E6POS: X 703.0705, Y -69.3124, Z -128.0150, A 0, B 90, C 0, E1 0, E2 0, E3 0, E4 0 } C_DIS
LIN{ E6POS: X 703.1278, Y -69.0963, Z -128.0150, A 0, B 90, C 0, E1 0, E2 0, E3 0, E4 0 } C_DIS
LIN{ E6POS: X 703.1910, Y -68.8829, Z -128.0150, A 0, B 90, C 0, E1 0, E2 0, E3 0, E4 0 } C_DIS
LIN{ E6POS: X 703.4360, Y -67.9134, Z -128.0150, A 0, B 90, C 0, E1 0, E2 0, E3 0, E4 0 } C_DIS
LIN{ E6POS: X 703.4975, Y -67.6700, Z -128.0150, A 0, B 90, C 0, E1 0, E2 0, E3 0, E4 0 } C_DIS
LIN{ E6POS: X 703.5593, Y -67.4497, Z -128.0150, A 0, B 90, C 0, E1 0, E2 0, E3 0, E4 0 } C_DIS
LIN{ E6POS: X 703.7865, Y -66.4759, Z -128.0150, A 0, B 90, C 0, E1 0, E2 0, E3 0, E4 0 } C_DIS
LIN{ E6POS: X 703.8524, Y -66.1933, Z -128.0150, A 0, B 90, C 0, E1 0, E2 0, E3 0, E4 0 } C_DIS
LIN{ E6POS: X 703.9118, Y -65.9608, Z -128.0150, A 0, B 90, C 0, E1 0, E2 0, E3 0, E4 0 } C_DIS
LIN{ E6POS: X 704.1259, Y -64.9840, Z -128.0150, A 0, B 90, C 0, E1 0, E2 0, E3 0, E4 0 } C_DIS
LIN{ E6POS: X 704.1900, Y -64.6919, Z -128.0150, A 0, B 90, C 0, E1 0, E2 0, E3 0, E4 0 } C_DIS
LIN{ E6POS: X 704.2474, Y -64.4539, Z -128.0150, A 0, B 90, C 0, E1 0, E2 0, E3 0, E4 0 } C_DIS
LIN{ E6POS: X 704.4528, Y -63.4752, Z -128.0150, A 0, B 90, C 0, E1 0, E2 0, E3 0, E4 0 } C_DIS
LIN{ E6POS: X 704.5101, Y -63.2020, Z -128.0150, A 0, B 90, C 0, E1 0, E2 0, E3 0, E4 0 } C_DIS
LIN{ E6POS: X 704.5653, Y -62.9658, Z -128.0150, A 0, B 90, C 0, E1 0, E2 0, E3 0, E4 0 } C_DIS
LIN{ E6POS: X 704.7658, Y -61.9861, Z -128.0150, A 0, B 90, C 0, E1 0, E2 0, E3 0, E4 0 } C_DIS
LIN{ E6POS: X 704.8117, Y -61.7620, Z -128.0150, A 0, B 90, C 0, E1 0, E2 0, E3 0, E4 0 } C_DIS
LIN{ E6POS: X 704.8648, Y -61.5343, Z -128.0150, A 0, B 90, C 0, E1 0, E2 0, E3 0, E4 0 } C_DIS
LIN{ E6POS: X 705.0646, Y -60.5545, Z -128.0150, A 0, B 90, C 0, E1 0, E2 0, E3 0, E4 0 } C_DIS
LIN{ E6POS: X 705.0946, Y -60.4074, Z -128.0150, A 0, B 90, C 0, E1 0, E2 0, E3 0, E4 0 } C_DIS
LIN{ E6POS: X 705.1457, Y -60.1954, Z -128.0150, A 0, B 90, C 0, E1 0, E2 0, E3 0, E4 0 } C_DIS
LIN{ E6POS: X 705.3408, Y -59.2146, Z -128.0150, A 0, B 90, C 0, E1 0, E2 0, E3 0, E4 0 } C_DIS
LIN{ E6POS: X 705.3619, Y -59.1087, Z -128.0150, A 0, B 90, C 0, E1 0, E2 0, E3 0, E4 0 } C_DIS
LIN{ E6POS: X 705.4114, Y -58.9045, Z -128.0150, A 0, B 90, C 0, E1 0, E2 0, E3 0, E4 0 } C_DIS
LIN{ E6POS: X 705.6004, Y -57.9226, Z -128.0150, A 0, B 90, C 0, E1 0, E2 0, E3 0, E4 0 } C_DIS
LIN{ E6POS: X 705.6206, Y -57.8175, Z -128.0150, A 0, B 90, C 0, E1 0, E2 0, E3 0, E4 0 } C_DIS
LIN{ E6POS: X 705.6685, Y -57.6134, Z -128.0150, A 0, B 90, C 0, E1 0, E2 0, E3 0, E4 0 } C_DIS
LIN{ E6POS: X 705.8488, Y -56.6298, Z -128.0150, A 0, B 90, C 0, E1 0, E2 0, E3 0, E4 0 } C_DIS
LIN{ E6POS: X 705.8747, Y -56.4887, Z -128.0150, A 0, B 90, C 0, E1 0, E2 0, E3 0, E4 0 } C_DIS
LIN{ E6POS: X 705.9213, Y -56.2770, Z -128.0150, A 0, B 90, C 0, E1 0, E2 0, E3 0, E4 0 } C_DIS
LIN{ E6POS: X 706.0912, Y -55.2915, Z -128.0150, A 0, B 90, C 0, E1 0, E2 0, E3 0, E4 0 } C_DIS
LIN{ E6POS: X 706.1287, Y -55.0741, Z -128.0150, A 0, B 90, C 0, E1 0, E2 0, E3 0, E4 0 } C_DIS
LIN{ E6POS: X 706.1744, Y -54.8471, Z -128.0150, A 0, B 90, C 0, E1 0, E2 0, E3 0, E4 0 } C_DIS
LIN{ E6POS: X 706.3377, Y -53.8605, Z -128.0150, A 0, B 90, C 0, E1 0, E2 0, E3 0, E4 0 } C_DIS
LIN{ E6POS: X 706.3798, Y -53.6060, Z -128.0150, A 0, B 90, C 0, E1 0, E2 0, E3 0, E4 0 } C_DIS
LIN{ E6POS: X 706.4244, Y -53.3711, Z -128.0150, A 0, B 90, C 0, E1 0, E2 0, E3 0, E4 0 } C_DIS
LIN{ E6POS: X 706.5826, Y -52.3837, Z -128.0150, A 0, B 90, C 0, E1 0, E2 0, E3 0, E4 0 } C_DIS
LIN{ E6POS: X 706.6232, Y -52.1306, Z -128.0150, A 0, B 90, C 0, E1 0, E2 0, E3 0, E4 0 } C_DIS
LIN{ E6POS: X 706.6667, Y -51.8958, Z -128.0150, A 0, B 90, C 0, E1 0, E2 0, E3 0, E4 0 } C_DIS
LIN{ E6POS: X 706.8227, Y -50.9080, Z -128.0150, A 0, B 90, C 0, E1 0, E2 0, E3 0, E4 0 } C_DIS
LIN{ E6POS: X 706.8566, Y -50.6935, Z -128.0150, A 0, B 90, C 0, E1 0, E2 0, E3 0, E4 0 } C_DIS
LIN{ E6POS: X 706.8988, Y -50.4665, Z -128.0150, A 0, B 90, C 0, E1 0, E2 0, E3 0, E4 0 } C_DIS
LIN{ E6POS: X 707.0541, Y -49.4787, Z -128.0150, A 0, B 90, C 0, E1 0, E2 0, E3 0, E4 0 } C_DIS
LIN{ E6POS: X 707.0755, Y -49.3431, Z -128.0150, A 0, B 90, C 0, E1 0, E2 0, E3 0, E4 0 } C_DIS
LIN{ E6POS: X 707.1165, Y -49.1316, Z -128.0150, A 0, B 90, C 0, E1 0, E2 0, E3 0, E4 0 } C_DIS
LIN{ E6POS: X 707.2723, Y -48.1438, Z -128.0150, A 0, B 90, C 0, E1 0, E2 0, E3 0, E4 0 } C_DIS
LIN{ E6POS: X 707.2808, Y -48.0898, Z -128.0150, A 0, B 90, C 0, E1 0, E2 0, E3 0, E4 0 } C_DIS
LIN{ E6POS: X 707.3205, Y -47.8922, Z -128.0150, A 0, B 90, C 0, E1 0, E2 0, E3 0, E4 0 } C_DIS
LIN{ E6POS: X 707.4730, Y -46.9393, Z -128.0150, A 0, B 90, C 0, E1 0, E2 0, E3 0, E4 0 } C_DIS
LIN{ E6POS: X 707.5112, Y -46.7541, Z -128.0150, A 0, B 90, C 0, E1 0, E2 0, E3 0, E4 0 } C_DIS
LIN{ E6POS: X 707.6786, Y -45.7683, Z -128.0150, A 0, B 90, C 0, E1 0, E2 0, E3 0, E4 0 } C_DIS
LIN{ E6POS: X 707.8461, Y -44.7824, Z -128.0150, A 0, B 90, C 0, E1 0, E2 0, E3 0, E4 0 } C_DIS
LIN{ E6POS: X 707.8481, Y -44.7710, Z -128.0150, A 0, B 90, C 0, E1 0, E2 0, E3 0, E4 0 } C_DIS
LIN{ E6POS: X 707.8844, Y -44.5968, Z -128.0150, A 0, B 90, C 0, E1 0, E2 0, E3 0, E4 0 } C_DIS
LIN{ E6POS: X 707.9190, Y -44.4318, Z -128.0150, A 0, B 90, C 0, E1 0, E2 0, E3 0, E4 0 } C_DIS
LIN{ E6POS: X 707.9523, Y -44.2686, Z -128.0150, A 0, B 90, C 0, E1 0, E2 0, E3 0, E4 0 } C_DIS
LIN{ E6POS: X 707.9846, Y -44.0994, Z -128.0150, A 0, B 90, C 0, E1 0, E2 0, E3 0, E4 0 } C_DIS
LIN{ E6POS: X 708.1476, Y -43.1128, Z -128.0150, A 0, B 90, C 0, E1 0, E2 0, E3 0, E4 0 } C_DIS
LIN{ E6POS: X 708.3054, Y -42.1575, Z -128.0150, A 0, B 90, C 0, E1 0, E2 0, E3 0, E4 0 } C_DIS
LIN{ E6POS: X 708.3377, Y -41.9745, Z -128.0150, A 0, B 90, C 0, E1 0, E2 0, E3 0, E4 0 } C_DIS
LIN{ E6POS: X 708.4739, Y -41.0052, Z -128.0150, A 0, B 90, C 0, E1 0, E2 0, E3 0, E4 0 } C_DIS
LIN{ E6POS: X 708.5064, Y -40.8008, Z -128.0150, A 0, B 90, C 0, E1 0, E2 0, E3 0, E4 0 } C_DIS
LIN{ E6POS: X 708.6346, Y -39.8091, Z -128.0150, A 0, B 90, C 0, E1 0, E2 0, E3 0, E4 0 } C_DIS
LIN{ E6POS: X 708.6439, Y -39.7375, Z -128.0150, A 0, B 90, C 0, E1 0, E2 0, E3 0, E4 0 } C_DIS
LIN{ E6POS: X 708.6762, Y -39.5203, Z -128.0150, A 0, B 90, C 0, E1 0, E2 0, E3 0, E4 0 } C_DIS
LIN{ E6POS: X 708.7974, Y -38.5277, Z -128.0150, A 0, B 90, C 0, E1 0, E2 0, E3 0, E4 0 } C_DIS
LIN{ E6POS: X 708.8119, Y -38.4085, Z -128.0150, A 0, B 90, C 0, E1 0, E2 0, E3 0, E4 0 } C_DIS
LIN{ E6POS: X 708.8437, Y -38.1866, Z -128.0150, A 0, B 90, C 0, E1 0, E2 0, E3 0, E4 0 } C_DIS
LIN{ E6POS: X 708.9587, Y -37.1932, Z -128.0150, A 0, B 90, C 0, E1 0, E2 0, E3 0, E4 0 } C_DIS
LIN{ E6POS: X 708.9726, Y -37.0734, Z -128.0150, A 0, B 90, C 0, E1 0, E2 0, E3 0, E4 0 } C_DIS
LIN{ E6POS: X 709.0032, Y -36.8555, Z -128.0150, A 0, B 90, C 0, E1 0, E2 0, E3 0, E4 0 } C_DIS
LIN{ E6POS: X 709.1118, Y -35.8614, Z -128.0150, A 0, B 90, C 0, E1 0, E2 0, E3 0, E4 0 } C_DIS
LIN{ E6POS: X 709.1201, Y -35.7858, Z -128.0150, A 0, B 90, C 0, E1 0, E2 0, E3 0, E4 0 } C_DIS
LIN{ E6POS: X 709.1492, Y -35.5800, Z -128.0150, A 0, B 90, C 0, E1 0, E2 0, E3 0, E4 0 } C_DIS
LIN{ E6POS: X 709.2520, Y -34.5853, Z -128.0150, A 0, B 90, C 0, E1 0, E2 0, E3 0, E4 0 } C_DIS
LIN{ E6POS: X 709.2581, Y -34.5262, Z -128.0150, A 0, B 90, C 0, E1 0, E2 0, E3 0, E4 0 } C_DIS
LIN{ E6POS: X 709.2861, Y -34.3260, Z -128.0150, A 0, B 90, C 0, E1 0, E2 0, E3 0, E4 0 } C_DIS
LIN{ E6POS: X 709.3847, Y -33.3309, Z -128.0150, A 0, B 90, C 0, E1 0, E2 0, E3 0, E4 0 } C_DIS
LIN{ E6POS: X 709.3921, Y -33.2555, Z -128.0150, A 0, B 90, C 0, E1 0, E2 0, E3 0, E4 0 } C_DIS
LIN{ E6POS: X 709.4191, Y -33.0539, Z -128.0150, A 0, B 90, C 0, E1 0, E2 0, E3 0, E4 0 } C_DIS
LIN{ E6POS: X 709.5129, Y -32.0583, Z -128.0150, A 0, B 90, C 0, E1 0, E2 0, E3 0, E4 0 } C_DIS
LIN{ E6POS: X 709.5243, Y -31.9377, Z -128.0150, A 0, B 90, C 0, E1 0, E2 0, E3 0, E4 0 } C_DIS
LIN{ E6POS: X 709.5507, Y -31.7280, Z -128.0150, A 0, B 90, C 0, E1 0, E2 0, E3 0, E4 0 } C_DIS
LIN{ E6POS: X 709.6417, Y -30.7321, Z -128.0150, A 0, B 90, C 0, E1 0, E2 0, E3 0, E4 0 } C_DIS
LIN{ E6POS: X 709.6597, Y -30.5353, Z -128.0150, A 0, B 90, C 0, E1 0, E2 0, E3 0, E4 0 } C_DIS
LIN{ E6POS: X 709.6858, Y -30.3103, Z -128.0150, A 0, B 90, C 0, E1 0, E2 0, E3 0, E4 0 } C_DIS
LIN{ E6POS: X 709.7741, Y -29.3142, Z -128.0150, A 0, B 90, C 0, E1 0, E2 0, E3 0, E4 0 } C_DIS
LIN{ E6POS: X 709.7949, Y -29.0801, Z -128.0150, A 0, B 90, C 0, E1 0, E2 0, E3 0, E4 0 } C_DIS
LIN{ E6POS: X 709.8208, Y -28.8477, Z -128.0150, A 0, B 90, C 0, E1 0, E2 0, E3 0, E4 0 } C_DIS
LIN{ E6POS: X 709.9065, Y -27.8514, Z -128.0150, A 0, B 90, C 0, E1 0, E2 0, E3 0, E4 0 } C_DIS
LIN{ E6POS: X 709.9266, Y -27.6182, Z -128.0150, A 0, B 90, C 0, E1 0, E2 0, E3 0, E4 0 } C_DIS
LIN{ E6POS: X 709.9516, Y -27.3858, Z -128.0150, A 0, B 90, C 0, E1 0, E2 0, E3 0, E4 0 } C_DIS
LIN{ E6POS: X 710.0338, Y -26.3892, Z -128.0150, A 0, B 90, C 0, E1 0, E2 0, E3 0, E4 0 } C_DIS
LIN{ E6POS: X 710.0498, Y -26.1950, Z -128.0150, A 0, B 90, C 0, E1 0, E2 0, E3 0, E4 0 } C_DIS
LIN{ E6POS: X 710.0741, Y -25.9704, Z -128.0150, A 0, B 90, C 0, E1 0, E2 0, E3 0, E4 0 } C_DIS
LIN{ E6POS: X 710.1527, Y -24.9735, Z -128.0150, A 0, B 90, C 0, E1 0, E2 0, E3 0, E4 0 } C_DIS
LIN{ E6POS: X 710.1618, Y -24.8575, Z -128.0150, A 0, B 90, C 0, E1 0, E2 0, E3 0, E4 0 } C_DIS
LIN{ E6POS: X 710.1849, Y -24.6482, Z -128.0150, A 0, B 90, C 0, E1 0, E2 0, E3 0, E4 0 } C_DIS
LIN{ E6POS: X 710.2590, Y -23.6510, Z -128.0150, A 0, B 90, C 0, E1 0, E2 0, E3 0, E4 0 } C_DIS
LIN{ E6POS: X 710.2640, Y -23.5841, Z -128.0150, A 0, B 90, C 0, E1 0, E2 0, E3 0, E4 0 } C_DIS
LIN{ E6POS: X 710.2860, Y -23.3851, Z -128.0150, A 0, B 90, C 0, E1 0, E2 0, E3 0, E4 0 } C_DIS
LIN{ E6POS: X 710.3556, Y -22.3875, Z -128.0150, A 0, B 90, C 0, E1 0, E2 0, E3 0, E4 0 } C_DIS
LIN{ E6POS: X 710.3590, Y -22.3383, Z -128.0150, A 0, B 90, C 0, E1 0, E2 0, E3 0, E4 0 } C_DIS
LIN{ E6POS: X 710.3796, Y -22.1445, Z -128.0150, A 0, B 90, C 0, E1 0, E2 0, E3 0, E4 0 } C_DIS
LIN{ E6POS: X 710.4457, Y -21.1467, Z -128.0150, A 0, B 90, C 0, E1 0, E2 0, E3 0, E4 0 } C_DIS
LIN{ E6POS: X 710.4496, Y -21.0881, Z -128.0150, A 0, B 90, C 0, E1 0, E2 0, E3 0, E4 0 } C_DIS
LIN{ E6POS: X 710.4690, Y -20.8945, Z -128.0150, A 0, B 90, C 0, E1 0, E2 0, E3 0, E4 0 } C_DIS
LIN{ E6POS: X 710.5322, Y -19.8965, Z -128.0150, A 0, B 90, C 0, E1 0, E2 0, E3 0, E4 0 } C_DIS
LIN{ E6POS: X 710.5385, Y -19.7969, Z -128.0150, A 0, B 90, C 0, E1 0, E2 0, E3 0, E4 0 } C_DIS
LIN{ E6POS: X 710.5564, Y -19.5986, Z -128.0150, A 0, B 90, C 0, E1 0, E2 0, E3 0, E4 0 } C_DIS
LIN{ E6POS: X 710.6170, Y -18.6004, Z -128.0150, A 0, B 90, C 0, E1 0, E2 0, E3 0, E4 0 } C_DIS
LIN{ E6POS: X 710.6249, Y -18.4709, Z -128.0150, A 0, B 90, C 0, E1 0, E2 0, E3 0, E4 0 } C_DIS
LIN{ E6POS: X 710.6416, Y -18.2689, Z -128.0150, A 0, B 90, C 0, E1 0, E2 0, E3 0, E4 0 } C_DIS
LIN{ E6POS: X 710.7017, Y -17.2707, Z -128.0150, A 0, B 90, C 0, E1 0, E2 0, E3 0, E4 0 } C_DIS
LIN{ E6POS: X 710.7107, Y -17.1205, Z -128.0150, A 0, B 90, C 0, E1 0, E2 0, E3 0, E4 0 } C_DIS
LIN{ E6POS: X 710.7267, Y -16.9161, Z -128.0150, A 0, B 90, C 0, E1 0, E2 0, E3 0, E4 0 } C_DIS
LIN{ E6POS: X 710.7895, Y -15.9181, Z -128.0150, A 0, B 90, C 0, E1 0, E2 0, E3 0, E4 0 } C_DIS
LIN{ E6POS: X 710.8352, Y -15.1932, Z -128.0150, A 0, B 90, C 0, E1 0, E2 0, E3 0, E4 0 } C_DIS
LIN{ E6POS: X 710.8633, Y -14.8566, Z -128.0150, A 0, B 90, C 0, E1 0, E2 0, E3 0, E4 0 } C_DIS
LIN{ E6POS: X 710.9199, Y -13.8582, Z -128.0150, A 0, B 90, C 0, E1 0, E2 0, E3 0, E4 0 } C_DIS
LIN{ E6POS: X 710.9765, Y -12.8598, Z -128.0150, A 0, B 90, C 0, E1 0, E2 0, E3 0, E4 0 } C_DIS
LIN{ E6POS: X 710.9792, Y -12.8129, Z -128.0150, A 0, B 90, C 0, E1 0, E2 0, E3 0, E4 0 } C_DIS
LIN{ E6POS: X 711.0177, Y -12.4012, Z -128.0150, A 0, B 90, C 0, E1 0, E2 0, E3 0, E4 0 } C_DIS
LIN{ E6POS: X 711.0670, Y -11.4099, Z -128.0150, A 0, B 90, C 0, E1 0, E2 0, E3 0, E4 0 } C_DIS
LIN{ E6POS: X 711.0833, Y -11.2230, Z -128.0150, A 0, B 90, C 0, E1 0, E2 0, E3 0, E4 0 } C_DIS
LIN{ E6POS: X 711.1314, Y -10.2242, Z -128.0150, A 0, B 90, C 0, E1 0, E2 0, E3 0, E4 0 } C_DIS
LIN{ E6POS: X 711.1363, Y -10.1219, Z -128.0150, A 0, B 90, C 0, E1 0, E2 0, E3 0, E4 0 } C_DIS
LIN{ E6POS: X 711.1527, Y -9.9150, Z -128.0150, A 0, B 90, C 0, E1 0, E2 0, E3 0, E4 0 } C_DIS
LIN{ E6POS: X 711.1999, Y -8.9161, Z -128.0150, A 0, B 90, C 0, E1 0, E2 0, E3 0, E4 0 } C_DIS
LIN{ E6POS: X 711.2082, Y -8.7396, Z -128.0150, A 0, B 90, C 0, E1 0, E2 0, E3 0, E4 0 } C_DIS
LIN{ E6POS: X 711.2242, Y -8.5181, Z -128.0150, A 0, B 90, C 0, E1 0, E2 0, E3 0, E4 0 } C_DIS
LIN{ E6POS: X 711.2705, Y -7.5192, Z -128.0150, A 0, B 90, C 0, E1 0, E2 0, E3 0, E4 0 } C_DIS
LIN{ E6POS: X 711.2804, Y -7.3063, Z -128.0150, A 0, B 90, C 0, E1 0, E2 0, E3 0, E4 0 } C_DIS
LIN{ E6POS: X 711.2958, Y -7.0777, Z -128.0150, A 0, B 90, C 0, E1 0, E2 0, E3 0, E4 0 } C_DIS
LIN{ E6POS: X 711.3398, Y -6.0787, Z -128.0150, A 0, B 90, C 0, E1 0, E2 0, E3 0, E4 0 } C_DIS
LIN{ E6POS: X 711.3491, Y -5.8676, Z -128.0150, A 0, B 90, C 0, E1 0, E2 0, E3 0, E4 0 } C_DIS
LIN{ E6POS: X 711.3644, Y -5.6392, Z -128.0150, A 0, B 90, C 0, E1 0, E2 0, E3 0, E4 0 } C_DIS
LIN{ E6POS: X 711.4075, Y -4.6401, Z -128.0150, A 0, B 90, C 0, E1 0, E2 0, E3 0, E4 0 } C_DIS
LIN{ E6POS: X 711.4149, Y -4.4675, Z -128.0150, A 0, B 90, C 0, E1 0, E2 0, E3 0, E4 0 } C_DIS
LIN{ E6POS: X 711.4299, Y -4.2466, Z -128.0150, A 0, B 90, C 0, E1 0, E2 0, E3 0, E4 0 } C_DIS
LIN{ E6POS: X 711.4710, Y -3.2475, Z -128.0150, A 0, B 90, C 0, E1 0, E2 0, E3 0, E4 0 } C_DIS
LIN{ E6POS: X 711.4749, Y -3.1518, Z -128.0150, A 0, B 90, C 0, E1 0, E2 0, E3 0, E4 0 } C_DIS
LIN{ E6POS: X 711.4899, Y -2.9459, Z -128.0150, A 0, B 90, C 0, E1 0, E2 0, E3 0, E4 0 } C_DIS
LIN{ E6POS: X 711.5290, Y -1.9467, Z -128.0150, A 0, B 90, C 0, E1 0, E2 0, E3 0, E4 0 } C_DIS
LIN{ E6POS: X 711.5313, Y -1.8901, Z -128.0150, A 0, B 90, C 0, E1 0, E2 0, E3 0, E4 0 } C_DIS
LIN{ E6POS: X 711.5460, Y -1.6916, Z -128.0150, A 0, B 90, C 0, E1 0, E2 0, E3 0, E4 0 } C_DIS
LIN{ E6POS: X 711.5834, Y -0.6923, Z -128.0150, A 0, B 90, C 0, E1 0, E2 0, E3 0, E4 0 } C_DIS
LIN{ E6POS: X 711.5855, Y -0.6370, Z -128.0150, A 0, B 90, C 0, E1 0, E2 0, E3 0, E4 0 } C_DIS
LIN{ E6POS: X 711.5999, Y -0.4389, Z -128.0150, A 0, B 90, C 0, E1 0, E2 0, E3 0, E4 0 } C_DIS
LIN{ E6POS: X 711.6364, Y 0.5604, Z -128.0150, A 0, B 90, C 0, E1 0, E2 0, E3 0, E4 0 } C_DIS
LIN{ E6POS: X 711.6397, Y 0.6506, Z -128.0150, A 0, B 90, C 0, E1 0, E2 0, E3 0, E4 0 } C_DIS
LIN{ E6POS: X 711.6537, Y 0.8556, Z -128.0150, A 0, B 90, C 0, E1 0, E2 0, E3 0, E4 0 } C_DIS
LIN{ E6POS: X 711.6893, Y 1.8550, Z -128.0150, A 0, B 90, C 0, E1 0, E2 0, E3 0, E4 0 } C_DIS
LIN{ E6POS: X 711.6952, Y 2.0197, Z -128.0150, A 0, B 90, C 0, E1 0, E2 0, E3 0, E4 0 } C_DIS
LIN{ E6POS: X 711.7084, Y 2.2387, Z -128.0150, A 0, B 90, C 0, E1 0, E2 0, E3 0, E4 0 } C_DIS
LIN{ E6POS: X 711.7446, Y 3.2381, Z -128.0150, A 0, B 90, C 0, E1 0, E2 0, E3 0, E4 0 } C_DIS
LIN{ E6POS: X 711.7519, Y 3.4380, Z -128.0150, A 0, B 90, C 0, E1 0, E2 0, E3 0, E4 0 } C_DIS
LIN{ E6POS: X 711.7647, Y 3.6642, Z -128.0150, A 0, B 90, C 0, E1 0, E2 0, E3 0, E4 0 } C_DIS
LIN{ E6POS: X 711.7994, Y 4.6636, Z -128.0150, A 0, B 90, C 0, E1 0, E2 0, E3 0, E4 0 } C_DIS
LIN{ E6POS: X 711.8063, Y 4.8623, Z -128.0150, A 0, B 90, C 0, E1 0, E2 0, E3 0, E4 0 } C_DIS
LIN{ E6POS: X 711.8190, Y 5.0881, Z -128.0150, A 0, B 90, C 0, E1 0, E2 0, E3 0, E4 0 } C_DIS
LIN{ E6POS: X 711.8531, Y 6.0876, Z -128.0150, A 0, B 90, C 0, E1 0, E2 0, E3 0, E4 0 } C_DIS
LIN{ E6POS: X 711.8585, Y 6.2476, Z -128.0150, A 0, B 90, C 0, E1 0, E2 0, E3 0, E4 0 } C_DIS
LIN{ E6POS: X 711.8713, Y 6.4660, Z -128.0150, A 0, B 90, C 0, E1 0, E2 0, E3 0, E4 0 } C_DIS
LIN{ E6POS: X 711.9051, Y 7.4654, Z -128.0150, A 0, B 90, C 0, E1 0, E2 0, E3 0, E4 0 } C_DIS
LIN{ E6POS: X 711.9079, Y 7.5495, Z -128.0150, A 0, B 90, C 0, E1 0, E2 0, E3 0, E4 0 } C_DIS
LIN{ E6POS: X 711.9212, Y 7.7534, Z -128.0150, A 0, B 90, C 0, E1 0, E2 0, E3 0, E4 0 } C_DIS
LIN{ E6POS: X 711.9534, Y 8.7529, Z -128.0150, A 0, B 90, C 0, E1 0, E2 0, E3 0, E4 0 } C_DIS
LIN{ E6POS: X 711.9548, Y 8.7977, Z -128.0150, A 0, B 90, C 0, E1 0, E2 0, E3 0, E4 0 } C_DIS
LIN{ E6POS: X 711.9681, Y 8.9941, Z -128.0150, A 0, B 90, C 0, E1 0, E2 0, E3 0, E4 0 } C_DIS
LIN{ E6POS: X 712.0007, Y 9.9935, Z -128.0150, A 0, B 90, C 0, E1 0, E2 0, E3 0, E4 0 } C_DIS
LIN{ E6POS: X 712.0021, Y 10.0365, Z -128.0150, A 0, B 90, C 0, E1 0, E2 0, E3 0, E4 0 } C_DIS
LIN{ E6POS: X 712.0153, Y 10.2325, Z -128.0150, A 0, B 90, C 0, E1 0, E2 0, E3 0, E4 0 } C_DIS
LIN{ E6POS: X 712.0470, Y 11.2320, Z -128.0150, A 0, B 90, C 0, E1 0, E2 0, E3 0, E4 0 } C_DIS
LIN{ E6POS: X 712.0495, Y 11.3097, Z -128.0150, A 0, B 90, C 0, E1 0, E2 0, E3 0, E4 0 } C_DIS
LIN{ E6POS: X 712.0624, Y 11.5124, Z -128.0150, A 0, B 90, C 0, E1 0, E2 0, E3 0, E4 0 } C_DIS
LIN{ E6POS: X 712.0954, Y 12.5119, Z -128.0150, A 0, B 90, C 0, E1 0, E2 0, E3 0, E4 0 } C_DIS
LIN{ E6POS: X 712.1004, Y 12.6628, Z -128.0150, A 0, B 90, C 0, E1 0, E2 0, E3 0, E4 0 } C_DIS
LIN{ E6POS: X 712.1127, Y 12.8793, Z -128.0150, A 0, B 90, C 0, E1 0, E2 0, E3 0, E4 0 } C_DIS
LIN{ E6POS: X 712.1456, Y 13.8787, Z -128.0150, A 0, B 90, C 0, E1 0, E2 0, E3 0, E4 0 } C_DIS
LIN{ E6POS: X 712.1517, Y 14.0642, Z -128.0150, A 0, B 90, C 0, E1 0, E2 0, E3 0, E4 0 } C_DIS
LIN{ E6POS: X 712.1636, Y 14.2875, Z -128.0150, A 0, B 90, C 0, E1 0, E2 0, E3 0, E4 0 } C_DIS
LIN{ E6POS: X 712.1969, Y 15.2870, Z -128.0150, A 0, B 90, C 0, E1 0, E2 0, E3 0, E4 0 } C_DIS
LIN{ E6POS: X 712.2031, Y 15.4714, Z -128.0150, A 0, B 90, C 0, E1 0, E2 0, E3 0, E4 0 } C_DIS
LIN{ E6POS: X 712.2153, Y 15.6945, Z -128.0150, A 0, B 90, C 0, E1 0, E2 0, E3 0, E4 0 } C_DIS
LIN{ E6POS: X 712.2487, Y 16.6939, Z -128.0150, A 0, B 90, C 0, E1 0, E2 0, E3 0, E4 0 } C_DIS
LIN{ E6POS: X 712.2536, Y 16.8403, Z -128.0150, A 0, B 90, C 0, E1 0, E2 0, E3 0, E4 0 } C_DIS
LIN{ E6POS: X 712.2659, Y 17.0562, Z -128.0150, A 0, B 90, C 0, E1 0, E2 0, E3 0, E4 0 } C_DIS
LIN{ E6POS: X 712.2998, Y 18.0556, Z -128.0150, A 0, B 90, C 0, E1 0, E2 0, E3 0, E4 0 } C_DIS
LIN{ E6POS: X 712.3021, Y 18.1258, Z -128.0150, A 0, B 90, C 0, E1 0, E2 0, E3 0, E4 0 } C_DIS
LIN{ E6POS: X 712.3152, Y 18.3273, Z -128.0150, A 0, B 90, C 0, E1 0, E2 0, E3 0, E4 0 } C_DIS
LIN{ E6POS: X 712.3484, Y 19.3267, Z -128.0150, A 0, B 90, C 0, E1 0, E2 0, E3 0, E4 0 } C_DIS
LIN{ E6POS: X 712.3494, Y 19.3583, Z -128.0150, A 0, B 90, C 0, E1 0, E2 0, E3 0, E4 0 } C_DIS
LIN{ E6POS: X 712.3627, Y 19.5524, Z -128.0150, A 0, B 90, C 0, E1 0, E2 0, E3 0, E4 0 } C_DIS
LIN{ E6POS: X 712.3969, Y 20.5518, Z -128.0150, A 0, B 90, C 0, E1 0, E2 0, E3 0, E4 0 } C_DIS
LIN{ E6POS: X 712.3980, Y 20.5813, Z -128.0150, A 0, B 90, C 0, E1 0, E2 0, E3 0, E4 0 } C_DIS
LIN{ E6POS: X 712.4115, Y 20.7750, Z -128.0150, A 0, B 90, C 0, E1 0, E2 0, E3 0, E4 0 } C_DIS
LIN{ E6POS: X 712.4478, Y 21.7744, Z -128.0150, A 0, B 90, C 0, E1 0, E2 0, E3 0, E4 0 } C_DIS
LIN{ E6POS: X 712.4501, Y 21.8387, Z -128.0150, A 0, B 90, C 0, E1 0, E2 0, E3 0, E4 0 } C_DIS
LIN{ E6POS: X 712.4634, Y 22.0388, Z -128.0150, A 0, B 90, C 0, E1 0, E2 0, E3 0, E4 0 } C_DIS
LIN{ E6POS: X 712.5002, Y 23.0381, Z -128.0150, A 0, B 90, C 0, E1 0, E2 0, E3 0, E4 0 } C_DIS
LIN{ E6POS: X 712.5052, Y 23.1731, Z -128.0150, A 0, B 90, C 0, E1 0, E2 0, E3 0, E4 0 } C_DIS
LIN{ E6POS: X 712.5181, Y 23.3867, Z -128.0150, A 0, B 90, C 0, E1 0, E2 0, E3 0, E4 0 } C_DIS
LIN{ E6POS: X 712.5594, Y 24.3859, Z -128.0150, A 0, B 90, C 0, E1 0, E2 0, E3 0, E4 0 } C_DIS
LIN{ E6POS: X 712.5652, Y 24.5263, Z -128.0150, A 0, B 90, C 0, E1 0, E2 0, E3 0, E4 0 } C_DIS
LIN{ E6POS: X 712.5783, Y 24.7436, Z -128.0150, A 0, B 90, C 0, E1 0, E2 0, E3 0, E4 0 } C_DIS
LIN{ E6POS: X 712.6239, Y 25.7426, Z -128.0150, A 0, B 90, C 0, E1 0, E2 0, E3 0, E4 0 } C_DIS
LIN{ E6POS: X 712.6274, Y 25.8206, Z -128.0150, A 0, B 90, C 0, E1 0, E2 0, E3 0, E4 0 } C_DIS
LIN{ E6POS: X 712.6409, Y 26.0317, Z -128.0150, A 0, B 90, C 0, E1 0, E2 0, E3 0, E4 0 } C_DIS
LIN{ E6POS: X 712.7087, Y 27.0294, Z -128.0150, A 0, B 90, C 0, E1 0, E2 0, E3 0, E4 0 } C_DIS
LIN{ E6POS: X 712.7766, Y 28.0271, Z -128.0150, A 0, B 90, C 0, E1 0, E2 0, E3 0, E4 0 } C_DIS
LIN{ E6POS: X 712.7799, Y 28.0760, Z -128.0150, A 0, B 90, C 0, E1 0, E2 0, E3 0, E4 0 } C_DIS
LIN{ E6POS: X 712.7942, Y 28.2716, Z -128.0150, A 0, B 90, C 0, E1 0, E2 0, E3 0, E4 0 } C_DIS
LIN{ E6POS: X 712.8096, Y 28.4418, Z -128.0150, A 0, B 90, C 0, E1 0, E2 0, E3 0, E4 0 } C_DIS
LIN{ E6POS: X 712.8258, Y 28.6018, Z -128.0150, A 0, B 90, C 0, E1 0, E2 0, E3 0, E4 0 } C_DIS
LIN{ E6POS: X 712.8422, Y 28.7672, Z -128.0150, A 0, B 90, C 0, E1 0, E2 0, E3 0, E4 0 } C_DIS
LIN{ E6POS: X 712.9118, Y 29.7647, Z -128.0150, A 0, B 90, C 0, E1 0, E2 0, E3 0, E4 0 } C_DIS
LIN{ E6POS: X 712.9813, Y 30.7623, Z -128.0150, A 0, B 90, C 0, E1 0, E2 0, E3 0, E4 0 } C_DIS
LIN{ E6POS: X 712.9828, Y 30.7839, Z -128.0150, A 0, B 90, C 0, E1 0, E2 0, E3 0, E4 0 } C_DIS
LIN{ E6POS: X 712.9987, Y 30.9697, Z -128.0150, A 0, B 90, C 0, E1 0, E2 0, E3 0, E4 0 } C_DIS
LIN{ E6POS: X 713.0397, Y 31.9688, Z -128.0150, A 0, B 90, C 0, E1 0, E2 0, E3 0, E4 0 } C_DIS
LIN{ E6POS: X 713.0495, Y 32.2068, Z -128.0150, A 0, B 90, C 0, E1 0, E2 0, E3 0, E4 0 } C_DIS
LIN{ E6POS: X 713.0644, Y 32.4287, Z -128.0150, A 0, B 90, C 0, E1 0, E2 0, E3 0, E4 0 } C_DIS
LIN{ E6POS: X 713.0999, Y 33.4280, Z -128.0150, A 0, B 90, C 0, E1 0, E2 0, E3 0, E4 0 } C_DIS
LIN{ E6POS: X 713.1139, Y 33.8207, Z -128.0150, A 0, B 90, C 0, E1 0, E2 0, E3 0, E4 0 } C_DIS
LIN{ E6POS: X 713.1283, Y 34.0602, Z -128.0150, A 0, B 90, C 0, E1 0, E2 0, E3 0, E4 0 } C_DIS
LIN{ E6POS: X 713.1643, Y 35.0596, Z -128.0150, A 0, B 90, C 0, E1 0, E2 0, E3 0, E4 0 } C_DIS
LIN{ E6POS: X 713.1784, Y 35.4512, Z -128.0150, A 0, B 90, C 0, E1 0, E2 0, E3 0, E4 0 } C_DIS
LIN{ E6POS: X 713.1931, Y 35.6906, Z -128.0150, A 0, B 90, C 0, E1 0, E2 0, E3 0, E4 0 } C_DIS
LIN{ E6POS: X 713.2363, Y 36.6897, Z -128.0150, A 0, B 90, C 0, E1 0, E2 0, E3 0, E4 0 } C_DIS
LIN{ E6POS: X 713.2466, Y 36.9260, Z -128.0150, A 0, B 90, C 0, E1 0, E2 0, E3 0, E4 0 } C_DIS
LIN{ E6POS: X 713.2622, Y 37.1472, Z -128.0150, A 0, B 90, C 0, E1 0, E2 0, E3 0, E4 0 } C_DIS
LIN{ E6POS: X 713.3365, Y 38.1444, Z -128.0150, A 0, B 90, C 0, E1 0, E2 0, E3 0, E4 0 } C_DIS
LIN{ E6POS: X 713.3880, Y 38.8358, Z -128.0150, A 0, B 90, C 0, E1 0, E2 0, E3 0, E4 0 } C_DIS
LIN{ E6POS: X 713.4051, Y 39.0207, Z -128.0150, A 0, B 90, C 0, E1 0, E2 0, E3 0, E4 0 } C_DIS
LIN{ E6POS: X 713.4234, Y 39.1871, Z -128.0150, A 0, B 90, C 0, E1 0, E2 0, E3 0, E4 0 } C_DIS
LIN{ E6POS: X 713.4423, Y 39.3528, Z -128.0150, A 0, B 90, C 0, E1 0, E2 0, E3 0, E4 0 } C_DIS
LIN{ E6POS: X 713.5255, Y 40.3494, Z -128.0150, A 0, B 90, C 0, E1 0, E2 0, E3 0, E4 0 } C_DIS
LIN{ E6POS: X 713.5822, Y 41.0283, Z -128.0150, A 0, B 90, C 0, E1 0, E2 0, E3 0, E4 0 } C_DIS
LIN{ E6POS: X 713.6015, Y 41.2112, Z -128.0150, A 0, B 90, C 0, E1 0, E2 0, E3 0, E4 0 } C_DIS
LIN{ E6POS: X 713.6639, Y 42.2093, Z -128.0150, A 0, B 90, C 0, E1 0, E2 0, E3 0, E4 0 } C_DIS
LIN{ E6POS: X 713.6775, Y 42.4265, Z -128.0150, A 0, B 90, C 0, E1 0, E2 0, E3 0, E4 0 } C_DIS
LIN{ E6POS: X 713.6965, Y 42.6444, Z -128.0150, A 0, B 90, C 0, E1 0, E2 0, E3 0, E4 0 } C_DIS
LIN{ E6POS: X 713.7525, Y 43.6428, Z -128.0150, A 0, B 90, C 0, E1 0, E2 0, E3 0, E4 0 } C_DIS
LIN{ E6POS: X 713.7748, Y 44.0406, Z -128.0150, A 0, B 90, C 0, E1 0, E2 0, E3 0, E4 0 } C_DIS
LIN{ E6POS: X 713.7940, Y 44.2786, Z -128.0150, A 0, B 90, C 0, E1 0, E2 0, E3 0, E4 0 } C_DIS
LIN{ E6POS: X 713.8484, Y 45.2771, Z -128.0150, A 0, B 90, C 0, E1 0, E2 0, E3 0, E4 0 } C_DIS
LIN{ E6POS: X 713.8731, Y 45.7303, Z -128.0150, A 0, B 90, C 0, E1 0, E2 0, E3 0, E4 0 } C_DIS
LIN{ E6POS: X 713.8925, Y 45.9736, Z -128.0150, A 0, B 90, C 0, E1 0, E2 0, E3 0, E4 0 } C_DIS
LIN{ E6POS: X 713.9494, Y 46.9719, Z -128.0150, A 0, B 90, C 0, E1 0, E2 0, E3 0, E4 0 } C_DIS
LIN{ E6POS: X 713.9715, Y 47.3599, Z -128.0150, A 0, B 90, C 0, E1 0, E2 0, E3 0, E4 0 } C_DIS
LIN{ E6POS: X 713.9914, Y 47.5937, Z -128.0150, A 0, B 90, C 0, E1 0, E2 0, E3 0, E4 0 } C_DIS
LIN{ E6POS: X 714.0565, Y 48.5916, Z -128.0150, A 0, B 90, C 0, E1 0, E2 0, E3 0, E4 0 } C_DIS
LIN{ E6POS: X 714.0694, Y 48.7891, Z -128.0150, A 0, B 90, C 0, E1 0, E2 0, E3 0, E4 0 } C_DIS
LIN{ E6POS: X 714.0900, Y 48.9985, Z -128.0150, A 0, B 90, C 0, E1 0, E2 0, E3 0, E4 0 } C_DIS
LIN{ E6POS: X 714.1637, Y 49.9958, Z -128.0150, A 0, B 90, C 0, E1 0, E2 0, E3 0, E4 0 } C_DIS
LIN{ E6POS: X 714.1678, Y 50.0517, Z -128.0150, A 0, B 90, C 0, E1 0, E2 0, E3 0, E4 0 } C_DIS
LIN{ E6POS: X 714.1888, Y 50.2427, Z -128.0150, A 0, B 90, C 0, E1 0, E2 0, E3 0, E4 0 } C_DIS
LIN{ E6POS: X 714.2659, Y 51.2008, Z -128.0150, A 0, B 90, C 0, E1 0, E2 0, E3 0, E4 0 } C_DIS
LIN{ E6POS: X 714.2874, Y 51.3797, Z -128.0150, A 0, B 90, C 0, E1 0, E2 0, E3 0, E4 0 } C_DIS
LIN{ E6POS: X 714.3651, Y 52.3002, Z -128.0150, A 0, B 90, C 0, E1 0, E2 0, E3 0, E4 0 } C_DIS
LIN{ E6POS: X 714.4222, Y 52.4686, Z -128.0150, A 0, B 90, C 0, E1 0, E2 0, E3 0, E4 0 } C_DIS
LIN{ E6POS: X 715.2306, Y 52.2922, Z -128.0150, A 0, B 90, C 0, E1 0, E2 0, E3 0, E4 0 } C_DIS
LIN{ E6POS: X 716.1965, Y 52.0333, Z -128.0150, A 0, B 90, C 0, E1 0, E2 0, E3 0, E4 0 } C_DIS
LIN{ E6POS: X 717.1624, Y 51.7744, Z -128.0150, A 0, B 90, C 0, E1 0, E2 0, E3 0, E4 0 } C_DIS
LIN{ E6POS: X 717.6407, Y 51.6462, Z -128.0150, A 0, B 90, C 0, E1 0, E2 0, E3 0, E4 0 } C_DIS
LIN{ E6POS: X 718.1632, Y 51.5080, Z -128.0150, A 0, B 90, C 0, E1 0, E2 0, E3 0, E4 0 } C_DIS
LIN{ E6POS: X 719.1276, Y 51.2434, Z -128.0150, A 0, B 90, C 0, E1 0, E2 0, E3 0, E4 0 } C_DIS
LIN{ E6POS: X 720.0920, Y 50.9789, Z -128.0150, A 0, B 90, C 0, E1 0, E2 0, E3 0, E4 0 } C_DIS
LIN{ E6POS: X 721.0563, Y 50.7144, Z -128.0150, A 0, B 90, C 0, E1 0, E2 0, E3 0, E4 0 } C_DIS
LIN{ E6POS: X 722.0207, Y 50.4498, Z -128.0150, A 0, B 90, C 0, E1 0, E2 0, E3 0, E4 0 } C_DIS
LIN{ E6POS: X 722.9799, Y 50.1867, Z -128.0150, A 0, B 90, C 0, E1 0, E2 0, E3 0, E4 0 } C_DIS
LIN{ E6POS: X 723.8134, Y 49.9439, Z -128.0150, A 0, B 90, C 0, E1 0, E2 0, E3 0, E4 0 } C_DIS
LIN{ E6POS: X 724.7772, Y 49.6772, Z -128.0150, A 0, B 90, C 0, E1 0, E2 0, E3 0, E4 0 } C_DIS
LIN{ E6POS: X 725.7410, Y 49.4106, Z -128.0150, A 0, B 90, C 0, E1 0, E2 0, E3 0, E4 0 } C_DIS
LIN{ E6POS: X 726.7048, Y 49.1440, Z -128.0150, A 0, B 90, C 0, E1 0, E2 0, E3 0, E4 0 } C_DIS
LIN{ E6POS: X 727.6686, Y 48.8774, Z -128.0150, A 0, B 90, C 0, E1 0, E2 0, E3 0, E4 0 } C_DIS
LIN{ E6POS: X 728.6324, Y 48.6108, Z -128.0150, A 0, B 90, C 0, E1 0, E2 0, E3 0, E4 0 } C_DIS
LIN{ E6POS: X 729.5962, Y 48.3442, Z -128.0150, A 0, B 90, C 0, E1 0, E2 0, E3 0, E4 0 } C_DIS
LIN{ E6POS: X 730.5600, Y 48.0775, Z -128.0150, A 0, B 90, C 0, E1 0, E2 0, E3 0, E4 0 } C_DIS
LIN{ E6POS: X 731.5238, Y 47.8109, Z -128.0150, A 0, B 90, C 0, E1 0, E2 0, E3 0, E4 0 } C_DIS
LIN{ E6POS: X 731.8399, Y 47.7235, Z -128.0150, A 0, B 90, C 0, E1 0, E2 0, E3 0, E4 0 } C_DIS
LIN{ E6POS: X 732.7989, Y 47.4401, Z -128.0150, A 0, B 90, C 0, E1 0, E2 0, E3 0, E4 0 } C_DIS
LIN{ E6POS: X 733.2283, Y 47.3133, Z -128.0150, A 0, B 90, C 0, E1 0, E2 0, E3 0, E4 0 } C_DIS
LIN{ E6POS: X 734.1950, Y 47.0575, Z -128.0150, A 0, B 90, C 0, E1 0, E2 0, E3 0, E4 0 } C_DIS
LIN{ E6POS: X 735.1617, Y 46.8018, Z -128.0150, A 0, B 90, C 0, E1 0, E2 0, E3 0, E4 0 } C_DIS
LIN{ E6POS: X 736.1285, Y 46.5460, Z -128.0150, A 0, B 90, C 0, E1 0, E2 0, E3 0, E4 0 } C_DIS
LIN{ E6POS: X 737.0952, Y 46.2902, Z -128.0150, A 0, B 90, C 0, E1 0, E2 0, E3 0, E4 0 } C_DIS
LIN{ E6POS: X 738.0619, Y 46.0345, Z -128.0150, A 0, B 90, C 0, E1 0, E2 0, E3 0, E4 0 } C_DIS
LIN{ E6POS: X 739.0287, Y 45.7787, Z -128.0150, A 0, B 90, C 0, E1 0, E2 0, E3 0, E4 0 } C_DIS
LIN{ E6POS: X 739.9954, Y 45.5229, Z -128.0150, A 0, B 90, C 0, E1 0, E2 0, E3 0, E4 0 } C_DIS
LIN{ E6POS: X 740.9622, Y 45.2672, Z -128.0150, A 0, B 90, C 0, E1 0, E2 0, E3 0, E4 0 } C_DIS
LIN{ E6POS: X 741.9289, Y 45.0114, Z -128.0150, A 0, B 90, C 0, E1 0, E2 0, E3 0, E4 0 } C_DIS
LIN{ E6POS: X 742.8956, Y 44.7556, Z -128.0150, A 0, B 90, C 0, E1 0, E2 0, E3 0, E4 0 } C_DIS
LIN{ E6POS: X 743.1746, Y 44.6818, Z -128.0150, A 0, B 90, C 0, E1 0, E2 0, E3 0, E4 0 } C_DIS
LIN{ E6POS: X 744.1371, Y 44.4106, Z -128.0150, A 0, B 90, C 0, E1 0, E2 0, E3 0, E4 0 } C_DIS
LIN{ E6POS: X 744.9010, Y 44.1953, Z -128.0150, A 0, B 90, C 0, E1 0, E2 0, E3 0, E4 0 } C_DIS
LIN{ E6POS: X 745.8731, Y 43.9609, Z -128.0150, A 0, B 90, C 0, E1 0, E2 0, E3 0, E4 0 } C_DIS
LIN{ E6POS: X 746.8452, Y 43.7264, Z -128.0150, A 0, B 90, C 0, E1 0, E2 0, E3 0, E4 0 } C_DIS
LIN{ E6POS: X 747.8174, Y 43.4920, Z -128.0150, A 0, B 90, C 0, E1 0, E2 0, E3 0, E4 0 } C_DIS
LIN{ E6POS: X 748.7895, Y 43.2575, Z -128.0150, A 0, B 90, C 0, E1 0, E2 0, E3 0, E4 0 } C_DIS
LIN{ E6POS: X 749.7616, Y 43.0231, Z -128.0150, A 0, B 90, C 0, E1 0, E2 0, E3 0, E4 0 } C_DIS
LIN{ E6POS: X 750.7337, Y 42.7886, Z -128.0150, A 0, B 90, C 0, E1 0, E2 0, E3 0, E4 0 } C_DIS
LIN{ E6POS: X 751.7059, Y 42.5542, Z -128.0150, A 0, B 90, C 0, E1 0, E2 0, E3 0, E4 0 } C_DIS
LIN{ E6POS: X 752.6780, Y 42.3197, Z -128.0150, A 0, B 90, C 0, E1 0, E2 0, E3 0, E4 0 } C_DIS
LIN{ E6POS: X 753.6501, Y 42.0853, Z -128.0150, A 0, B 90, C 0, E1 0, E2 0, E3 0, E4 0 } C_DIS
LIN{ E6POS: X 754.6223, Y 41.8509, Z -128.0150, A 0, B 90, C 0, E1 0, E2 0, E3 0, E4 0 } C_DIS
LIN{ E6POS: X 755.4826, Y 41.6434, Z -128.0150, A 0, B 90, C 0, E1 0, E2 0, E3 0, E4 0 } C_DIS
LIN{ E6POS: X 756.4514, Y 41.3958, Z -128.0150, A 0, B 90, C 0, E1 0, E2 0, E3 0, E4 0 } C_DIS
LIN{ E6POS: X 757.3295, Y 41.1715, Z -128.0150, A 0, B 90, C 0, E1 0, E2 0, E3 0, E4 0 } C_DIS
LIN{ E6POS: X 758.3101, Y 40.9755, Z -128.0150, A 0, B 90, C 0, E1 0, E2 0, E3 0, E4 0 } C_DIS
LIN{ E6POS: X 759.2907, Y 40.7794, Z -128.0150, A 0, B 90, C 0, E1 0, E2 0, E3 0, E4 0 } C_DIS
LIN{ E6POS: X 760.2713, Y 40.5834, Z -128.0150, A 0, B 90, C 0, E1 0, E2 0, E3 0, E4 0 } C_DIS
LIN{ E6POS: X 761.2519, Y 40.3874, Z -128.0150, A 0, B 90, C 0, E1 0, E2 0, E3 0, E4 0 } C_DIS
LIN{ E6POS: X 762.2325, Y 40.1913, Z -128.0150, A 0, B 90, C 0, E1 0, E2 0, E3 0, E4 0 } C_DIS
LIN{ E6POS: X 763.2131, Y 39.9953, Z -128.0150, A 0, B 90, C 0, E1 0, E2 0, E3 0, E4 0 } C_DIS
LIN{ E6POS: X 764.1937, Y 39.7993, Z -128.0150, A 0, B 90, C 0, E1 0, E2 0, E3 0, E4 0 } C_DIS
LIN{ E6POS: X 765.1743, Y 39.6032, Z -128.0150, A 0, B 90, C 0, E1 0, E2 0, E3 0, E4 0 } C_DIS
LIN{ E6POS: X 766.1549, Y 39.4072, Z -128.0150, A 0, B 90, C 0, E1 0, E2 0, E3 0, E4 0 } C_DIS
LIN{ E6POS: X 767.1355, Y 39.2111, Z -128.0150, A 0, B 90, C 0, E1 0, E2 0, E3 0, E4 0 } C_DIS
LIN{ E6POS: X 767.2571, Y 39.1868, Z -128.0150, A 0, B 90, C 0, E1 0, E2 0, E3 0, E4 0 } C_DIS
LIN{ E6POS: X 768.2359, Y 38.9821, Z -128.0150, A 0, B 90, C 0, E1 0, E2 0, E3 0, E4 0 } C_DIS
LIN{ E6POS: X 769.0076, Y 38.8207, Z -128.0150, A 0, B 90, C 0, E1 0, E2 0, E3 0, E4 0 } C_DIS
LIN{ E6POS: X 770.0010, Y 38.7055, Z -128.0150, A 0, B 90, C 0, E1 0, E2 0, E3 0, E4 0 } C_DIS
LIN{ E6POS: X 770.9943, Y 38.5904, Z -128.0150, A 0, B 90, C 0, E1 0, E2 0, E3 0, E4 0 } C_DIS
LIN{ E6POS: X 771.9877, Y 38.4752, Z -128.0150, A 0, B 90, C 0, E1 0, E2 0, E3 0, E4 0 } C_DIS
LIN{ E6POS: X 772.9810, Y 38.3600, Z -128.0150, A 0, B 90, C 0, E1 0, E2 0, E3 0, E4 0 } C_DIS
LIN{ E6POS: X 773.9744, Y 38.2449, Z -128.0150, A 0, B 90, C 0, E1 0, E2 0, E3 0, E4 0 } C_DIS
LIN{ E6POS: X 774.9677, Y 38.1297, Z -128.0150, A 0, B 90, C 0, E1 0, E2 0, E3 0, E4 0 } C_DIS
LIN{ E6POS: X 775.9611, Y 38.0145, Z -128.0150, A 0, B 90, C 0, E1 0, E2 0, E3 0, E4 0 } C_DIS
LIN{ E6POS: X 776.9544, Y 37.8994, Z -128.0150, A 0, B 90, C 0, E1 0, E2 0, E3 0, E4 0 } C_DIS
LIN{ E6POS: X 776.9937, Y 37.8948, Z -128.0150, A 0, B 90, C 0, E1 0, E2 0, E3 0, E4 0 } C_DIS
LIN{ E6POS: X 777.9868, Y 37.7777, Z -128.0150, A 0, B 90, C 0, E1 0, E2 0, E3 0, E4 0 } C_DIS
LIN{ E6POS: X 778.4307, Y 37.7254, Z -128.0150, A 0, B 90, C 0, E1 0, E2 0, E3 0, E4 0 } C_DIS
LIN{ E6POS: X 779.4305, Y 37.7049, Z -128.0150, A 0, B 90, C 0, E1 0, E2 0, E3 0, E4 0 } C_DIS
LIN{ E6POS: X 780.4303, Y 37.6844, Z -128.0150, A 0, B 90, C 0, E1 0, E2 0, E3 0, E4 0 } C_DIS
LIN{ E6POS: X 781.4301, Y 37.6640, Z -128.0150, A 0, B 90, C 0, E1 0, E2 0, E3 0, E4 0 } C_DIS
LIN{ E6POS: X 782.4299, Y 37.6435, Z -128.0150, A 0, B 90, C 0, E1 0, E2 0, E3 0, E4 0 } C_DIS
LIN{ E6POS: X 783.4296, Y 37.6230, Z -128.0150, A 0, B 90, C 0, E1 0, E2 0, E3 0, E4 0 } C_DIS
LIN{ E6POS: X 784.4294, Y 37.6026, Z -128.0150, A 0, B 90, C 0, E1 0, E2 0, E3 0, E4 0 } C_DIS
LIN{ E6POS: X 784.9613, Y 37.5917, Z -128.0150, A 0, B 90, C 0, E1 0, E2 0, E3 0, E4 0 } C_DIS
LIN{ E6POS: X 785.9611, Y 37.5735, Z -128.0150, A 0, B 90, C 0, E1 0, E2 0, E3 0, E4 0 } C_DIS
LIN{ E6POS: X 786.1630, Y 37.5698, Z -128.0150, A 0, B 90, C 0, E1 0, E2 0, E3 0, E4 0 } C_DIS
LIN{ E6POS: X 787.1605, Y 37.6406, Z -128.0150, A 0, B 90, C 0, E1 0, E2 0, E3 0, E4 0 } C_DIS
LIN{ E6POS: X 788.1580, Y 37.7114, Z -128.0150, A 0, B 90, C 0, E1 0, E2 0, E3 0, E4 0 } C_DIS
LIN{ E6POS: X 789.1555, Y 37.7822, Z -128.0150, A 0, B 90, C 0, E1 0, E2 0, E3 0, E4 0 } C_DIS
LIN{ E6POS: X 790.1530, Y 37.8530, Z -128.0150, A 0, B 90, C 0, E1 0, E2 0, E3 0, E4 0 } C_DIS
LIN{ E6POS: X 791.1505, Y 37.9238, Z -128.0150, A 0, B 90, C 0, E1 0, E2 0, E3 0, E4 0 } C_DIS
LIN{ E6POS: X 791.7234, Y 37.9645, Z -128.0150, A 0, B 90, C 0, E1 0, E2 0, E3 0, E4 0 } C_DIS
LIN{ E6POS: X 792.7207, Y 38.0374, Z -128.0150, A 0, B 90, C 0, E1 0, E2 0, E3 0, E4 0 } C_DIS
LIN{ E6POS: X 792.7685, Y 38.0409, Z -128.0150, A 0, B 90, C 0, E1 0, E2 0, E3 0, E4 0 } C_DIS
LIN{ E6POS: X 793.7601, Y 38.1698, Z -128.0150, A 0, B 90, C 0, E1 0, E2 0, E3 0, E4 0 } C_DIS
LIN{ E6POS: X 794.7518, Y 38.2986, Z -128.0150, A 0, B 90, C 0, E1 0, E2 0, E3 0, E4 0 } C_DIS
LIN{ E6POS: X 795.7435, Y 38.4275, Z -128.0150, A 0, B 90, C 0, E1 0, E2 0, E3 0, E4 0 } C_DIS
LIN{ E6POS: X 796.7351, Y 38.5564, Z -128.0150, A 0, B 90, C 0, E1 0, E2 0, E3 0, E4 0 } C_DIS
LIN{ E6POS: X 797.7268, Y 38.6853, Z -128.0150, A 0, B 90, C 0, E1 0, E2 0, E3 0, E4 0 } C_DIS
LIN{ E6POS: X 797.8431, Y 38.7004, Z -128.0150, A 0, B 90, C 0, E1 0, E2 0, E3 0, E4 0 } C_DIS
LIN{ E6POS: X 798.8097, Y 38.8260, Z -128.0150, A 0, B 90, C 0, E1 0, E2 0, E3 0, E4 0 } C_DIS
LIN{ E6POS: X 798.7068, Y 37.8313, Z -128.0150, A 0, B 90, C 0, E1 0, E2 0, E3 0, E4 0 } C_DIS
LIN{ E6POS: X 798.6040, Y 36.8366, Z -128.0150, A 0, B 90, C 0, E1 0, E2 0, E3 0, E4 0 } C_DIS
LIN{ E6POS: X 798.5012, Y 35.8419, Z -128.0150, A 0, B 90, C 0, E1 0, E2 0, E3 0, E4 0 } C_DIS
LIN{ E6POS: X 798.3983, Y 34.8472, Z -128.0150, A 0, B 90, C 0, E1 0, E2 0, E3 0, E4 0 } C_DIS
LIN{ E6POS: X 798.2955, Y 33.8525, Z -128.0150, A 0, B 90, C 0, E1 0, E2 0, E3 0, E4 0 } C_DIS
LIN{ E6POS: X 798.1927, Y 32.8578, Z -128.0150, A 0, B 90, C 0, E1 0, E2 0, E3 0, E4 0 } C_DIS
LIN{ E6POS: X 798.0898, Y 31.8631, Z -128.0150, A 0, B 90, C 0, E1 0, E2 0, E3 0, E4 0 } C_DIS
LIN{ E6POS: X 797.9870, Y 30.8684, Z -128.0150, A 0, B 90, C 0, E1 0, E2 0, E3 0, E4 0 } C_DIS
LIN{ E6POS: X 797.8842, Y 29.8737, Z -128.0150, A 0, B 90, C 0, E1 0, E2 0, E3 0, E4 0 } C_DIS
LIN{ E6POS: X 797.7813, Y 28.8790, Z -128.0150, A 0, B 90, C 0, E1 0, E2 0, E3 0, E4 0 } C_DIS
LIN{ E6POS: X 797.6785, Y 27.8843, Z -128.0150, A 0, B 90, C 0, E1 0, E2 0, E3 0, E4 0 } C_DIS
LIN{ E6POS: X 797.5757, Y 26.8896, Z -128.0150, A 0, B 90, C 0, E1 0, E2 0, E3 0, E4 0 } C_DIS
LIN{ E6POS: X 797.4728, Y 25.8949, Z -128.0150, A 0, B 90, C 0, E1 0, E2 0, E3 0, E4 0 } C_DIS
LIN{ E6POS: X 797.3924, Y 25.1164, Z -128.0150, A 0, B 90, C 0, E1 0, E2 0, E3 0, E4 0 } C_DIS
LIN{ E6POS: X 797.2895, Y 24.1217, Z -128.0150, A 0, B 90, C 0, E1 0, E2 0, E3 0, E4 0 } C_DIS
LIN{ E6POS: X 797.1867, Y 23.1270, Z -128.0150, A 0, B 90, C 0, E1 0, E2 0, E3 0, E4 0 } C_DIS
LIN{ E6POS: X 797.1224, Y 22.5051, Z -128.0150, A 0, B 90, C 0, E1 0, E2 0, E3 0, E4 0 } C_DIS
LIN{ E6POS: X 797.0002, Y 21.5126, Z -128.0150, A 0, B 90, C 0, E1 0, E2 0, E3 0, E4 0 } C_DIS
LIN{ E6POS: X 796.8780, Y 20.5201, Z -128.0150, A 0, B 90, C 0, E1 0, E2 0, E3 0, E4 0 } C_DIS
LIN{ E6POS: X 796.7559, Y 19.5276, Z -128.0150, A 0, B 90, C 0, E1 0, E2 0, E3 0, E4 0 } C_DIS
LIN{ E6POS: X 796.6337, Y 18.5351, Z -128.0150, A 0, B 90, C 0, E1 0, E2 0, E3 0, E4 0 } C_DIS
LIN{ E6POS: X 796.5115, Y 17.5426, Z -128.0150, A 0, B 90, C 0, E1 0, E2 0, E3 0, E4 0 } C_DIS
LIN{ E6POS: X 796.3893, Y 16.5500, Z -128.0150, A 0, B 90, C 0, E1 0, E2 0, E3 0, E4 0 } C_DIS
LIN{ E6POS: X 796.2672, Y 15.5575, Z -128.0150, A 0, B 90, C 0, E1 0, E2 0, E3 0, E4 0 } C_DIS
LIN{ E6POS: X 796.1450, Y 14.5650, Z -128.0150, A 0, B 90, C 0, E1 0, E2 0, E3 0, E4 0 } C_DIS
LIN{ E6POS: X 796.0228, Y 13.5725, Z -128.0150, A 0, B 90, C 0, E1 0, E2 0, E3 0, E4 0 } C_DIS
LIN{ E6POS: X 795.9006, Y 12.5800, Z -128.0150, A 0, B 90, C 0, E1 0, E2 0, E3 0, E4 0 } C_DIS
LIN{ E6POS: X 795.7785, Y 11.5875, Z -128.0150, A 0, B 90, C 0, E1 0, E2 0, E3 0, E4 0 } C_DIS
LIN{ E6POS: X 795.6563, Y 10.5950, Z -128.0150, A 0, B 90, C 0, E1 0, E2 0, E3 0, E4 0 } C_DIS
LIN{ E6POS: X 795.5548, Y 9.7708, Z -128.0150, A 0, B 90, C 0, E1 0, E2 0, E3 0, E4 0 } C_DIS
LIN{ E6POS: X 795.4326, Y 8.7783, Z -128.0150, A 0, B 90, C 0, E1 0, E2 0, E3 0, E4 0 } C_DIS
LIN{ E6POS: X 795.3105, Y 7.7858, Z -128.0150, A 0, B 90, C 0, E1 0, E2 0, E3 0, E4 0 } C_DIS
LIN{ E6POS: X 795.2562, Y 7.3452, Z -126.0150, A 0, B 90, C 0, E1 0, E2 0, E3 0, E4 0 } C_DIS
LIN{ E6POS: X 795.0854, Y 6.3599, Z -126.0150, A 0, B 90, C 0, E1 0, E2 0, E3 0, E4 0 } C_DIS
LIN{ E6POS: X 794.9146, Y 5.3746, Z -126.0150, A 0, B 90, C 0, E1 0, E2 0, E3 0, E4 0 } C_DIS
LIN{ E6POS: X 794.7438, Y 4.3893, Z -126.0150, A 0, B 90, C 0, E1 0, E2 0, E3 0, E4 0 } C_DIS
LIN{ E6POS: X 794.5730, Y 3.4040, Z -126.0150, A 0, B 90, C 0, E1 0, E2 0, E3 0, E4 0 } C_DIS
LIN{ E6POS: X 794.4021, Y 2.4187, Z -126.0150, A 0, B 90, C 0, E1 0, E2 0, E3 0, E4 0 } C_DIS
LIN{ E6POS: X 794.2313, Y 1.4334, Z -126.0150, A 0, B 90, C 0, E1 0, E2 0, E3 0, E4 0 } C_DIS
LIN{ E6POS: X 794.0605, Y 0.4481, Z -126.0150, A 0, B 90, C 0, E1 0, E2 0, E3 0, E4 0 } C_DIS
LIN{ E6POS: X 793.8897, Y -0.5372, Z -126.0150, A 0, B 90, C 0, E1 0, E2 0, E3 0, E4 0 } C_DIS
LIN{ E6POS: X 793.7189, Y -1.5225, Z -126.0150, A 0, B 90, C 0, E1 0, E2 0, E3 0, E4 0 } C_DIS
LIN{ E6POS: X 793.5481, Y -2.5078, Z -126.0150, A 0, B 90, C 0, E1 0, E2 0, E3 0, E4 0 } C_DIS
LIN{ E6POS: X 793.3772, Y -3.4931, Z -126.0150, A 0, B 90, C 0, E1 0, E2 0, E3 0, E4 0 } C_DIS
LIN{ E6POS: X 793.2090, Y -4.4632, Z -126.0150, A 0, B 90, C 0, E1 0, E2 0, E3 0, E4 0 } C_DIS
LIN{ E6POS: X 793.0382, Y -5.4485, Z -126.0150, A 0, B 90, C 0, E1 0, E2 0, E3 0, E4 0 } C_DIS
LIN{ E6POS: X 793.0310, Y -5.4900, Z -126.0150, A 0, B 90, C 0, E1 0, E2 0, E3 0, E4 0 } C_DIS
LIN{ E6POS: X 792.7476, Y -6.4490, Z -126.0150, A 0, B 90, C 0, E1 0, E2 0, E3 0, E4 0 } C_DIS
LIN{ E6POS: X 792.4642, Y -7.4080, Z -126.0150, A 0, B 90, C 0, E1 0, E2 0, E3 0, E4 0 } C_DIS
LIN{ E6POS: X 792.1808, Y -8.3670, Z -126.0150, A 0, B 90, C 0, E1 0, E2 0, E3 0, E4 0 } C_DIS
LIN{ E6POS: X 791.8974, Y -9.3260, Z -126.0150, A 0, B 90, C 0, E1 0, E2 0, E3 0, E4 0 } C_DIS
LIN{ E6POS: X 791.6139, Y -10.2850, Z -126.0150, A 0, B 90, C 0, E1 0, E2 0, E3 0, E4 0 } C_DIS
LIN{ E6POS: X 791.3305, Y -11.2440, Z -126.0150, A 0, B 90, C 0, E1 0, E2 0, E3 0, E4 0 } C_DIS
LIN{ E6POS: X 791.0471, Y -12.2030, Z -126.0150, A 0, B 90, C 0, E1 0, E2 0, E3 0, E4 0 } C_DIS
LIN{ E6POS: X 790.7637, Y -13.1620, Z -126.0150, A 0, B 90, C 0, E1 0, E2 0, E3 0, E4 0 } C_DIS
LIN{ E6POS: X 790.4892, Y -14.0908, Z -126.0150, A 0, B 90, C 0, E1 0, E2 0, E3 0, E4 0 } C_DIS
LIN{ E6POS: X 790.2681, Y -14.8387, Z -126.0150, A 0, B 90, C 0, E1 0, E2 0, E3 0, E4 0 } C_DIS
LIN{ E6POS: X 789.6733, Y -15.6426, Z -126.0150, A 0, B 90, C 0, E1 0, E2 0, E3 0, E4 0 } C_DIS
LIN{ E6POS: X 789.0784, Y -16.4464, Z -126.0150, A 0, B 90, C 0, E1 0, E2 0, E3 0, E4 0 } C_DIS
LIN{ E6POS: X 788.4835, Y -17.2502, Z -126.0150, A 0, B 90, C 0, E1 0, E2 0, E3 0, E4 0 } C_DIS
LIN{ E6POS: X 787.8887, Y -18.0540, Z -126.0150, A 0, B 90, C 0, E1 0, E2 0, E3 0, E4 0 } C_DIS
LIN{ E6POS: X 787.2938, Y -18.8579, Z -126.0150, A 0, B 90, C 0, E1 0, E2 0, E3 0, E4 0 } C_DIS
LIN{ E6POS: X 787.0668, Y -19.1646, Z -126.0150, A 0, B 90, C 0, E1 0, E2 0, E3 0, E4 0 } C_DIS
LIN{ E6POS: X 786.7884, Y -19.5408, Z -126.0150, A 0, B 90, C 0, E1 0, E2 0, E3 0, E4 0 } C_DIS
LIN{ E6POS: X 785.8324, Y -19.8339, Z -126.0150, A 0, B 90, C 0, E1 0, E2 0, E3 0, E4 0 } C_DIS
LIN{ E6POS: X 784.8763, Y -20.1271, Z -126.0150, A 0, B 90, C 0, E1 0, E2 0, E3 0, E4 0 } C_DIS
LIN{ E6POS: X 783.9202, Y -20.4202, Z -126.0150, A 0, B 90, C 0, E1 0, E2 0, E3 0, E4 0 } C_DIS
LIN{ E6POS: X 782.9642, Y -20.7133, Z -126.0150, A 0, B 90, C 0, E1 0, E2 0, E3 0, E4 0 } C_DIS
LIN{ E6POS: X 782.7712, Y -20.7725, Z -126.0150, A 0, B 90, C 0, E1 0, E2 0, E3 0, E4 0 } C_DIS
LIN{ E6POS: X 782.4265, Y -20.8798, Z -126.0150, A 0, B 90, C 0, E1 0, E2 0, E3 0, E4 0 } C_DIS
LIN{ E6POS: X 782.0068, Y -20.8212, Z -126.0150, A 0, B 90, C 0, E1 0, E2 0, E3 0, E4 0 } C_DIS
LIN{ E6POS: X 781.0159, Y -20.6863, Z -126.0150, A 0, B 90, C 0, E1 0, E2 0, E3 0, E4 0 } C_DIS
LIN{ E6POS: X 780.0251, Y -20.5514, Z -126.0150, A 0, B 90, C 0, E1 0, E2 0, E3 0, E4 0 } C_DIS
LIN{ E6POS: X 779.0342, Y -20.4165, Z -126.0150, A 0, B 90, C 0, E1 0, E2 0, E3 0, E4 0 } C_DIS
LIN{ E6POS: X 778.0434, Y -20.2816, Z -126.0150, A 0, B 90, C 0, E1 0, E2 0, E3 0, E4 0 } C_DIS
LIN{ E6POS: X 777.0525, Y -20.1467, Z -126.0150, A 0, B 90, C 0, E1 0, E2 0, E3 0, E4 0 } C_DIS
LIN{ E6POS: X 777.0183, Y -20.1420, Z -126.0150, A 0, B 90, C 0, E1 0, E2 0, E3 0, E4 0 } C_DIS
LIN{ E6POS: X 776.5146, Y -20.0205, Z -126.0150, A 0, B 90, C 0, E1 0, E2 0, E3 0, E4 0 } C_DIS
LIN{ E6POS: X 775.5400, Y -19.7965, Z -126.0150, A 0, B 90, C 0, E1 0, E2 0, E3 0, E4 0 } C_DIS
LIN{ E6POS: X 774.5654, Y -19.5724, Z -126.0150, A 0, B 90, C 0, E1 0, E2 0, E3 0, E4 0 } C_DIS
LIN{ E6POS: X 773.5909, Y -19.3483, Z -126.0150, A 0, B 90, C 0, E1 0, E2 0, E3 0, E4 0 } C_DIS
LIN{ E6POS: X 772.6163, Y -19.1242, Z -126.0150, A 0, B 90, C 0, E1 0, E2 0, E3 0, E4 0 } C_DIS
LIN{ E6POS: X 771.6417, Y -18.9001, Z -126.0150, A 0, B 90, C 0, E1 0, E2 0, E3 0, E4 0 } C_DIS
LIN{ E6POS: X 770.6672, Y -18.6760, Z -126.0150, A 0, B 90, C 0, E1 0, E2 0, E3 0, E4 0 } C_DIS
LIN{ E6POS: X 770.3993, Y -18.6144, Z -126.0150, A 0, B 90, C 0, E1 0, E2 0, E3 0, E4 0 } C_DIS
LIN{ E6POS: X 769.8028, Y -18.5330, Z -126.0150, A 0, B 90, C 0, E1 0, E2 0, E3 0, E4 0 } C_DIS
LIN{ E6POS: X 768.8110, Y -18.4053, Z -126.0150, A 0, B 90, C 0, E1 0, E2 0, E3 0, E4 0 } C_DIS
LIN{ E6POS: X 767.8191, Y -18.2777, Z -126.0150, A 0, B 90, C 0, E1 0, E2 0, E3 0, E4 0 } C_DIS
LIN{ E6POS: X 766.8273, Y -18.1500, Z -126.0150, A 0, B 90, C 0, E1 0, E2 0, E3 0, E4 0 } C_DIS
LIN{ E6POS: X 765.8355, Y -18.0224, Z -126.0150, A 0, B 90, C 0, E1 0, E2 0, E3 0, E4 0 } C_DIS
LIN{ E6POS: X 764.8437, Y -17.8947, Z -126.0150, A 0, B 90, C 0, E1 0, E2 0, E3 0, E4 0 } C_DIS
LIN{ E6POS: X 763.8519, Y -17.7671, Z -126.0150, A 0, B 90, C 0, E1 0, E2 0, E3 0, E4 0 } C_DIS
LIN{ E6POS: X 762.8600, Y -17.6394, Z -126.0150, A 0, B 90, C 0, E1 0, E2 0, E3 0, E4 0 } C_DIS
LIN{ E6POS: X 762.4043, Y -17.5808, Z -126.0150, A 0, B 90, C 0, E1 0, E2 0, E3 0, E4 0 } C_DIS
LIN{ E6POS: X 761.7840, Y -17.5374, Z -126.0150, A 0, B 90, C 0, E1 0, E2 0, E3 0, E4 0 } C_DIS
LIN{ E6POS: X 760.7862, Y -17.4702, Z -126.0150, A 0, B 90, C 0, E1 0, E2 0, E3 0, E4 0 } C_DIS
LIN{ E6POS: X 759.7885, Y -17.4031, Z -126.0150, A 0, B 90, C 0, E1 0, E2 0, E3 0, E4 0 } C_DIS
LIN{ E6POS: X 758.7907, Y -17.3360, Z -126.0150, A 0, B 90, C 0, E1 0, E2 0, E3 0, E4 0 } C_DIS
LIN{ E6POS: X 757.7930, Y -17.2689, Z -126.0150, A 0, B 90, C 0, E1 0, E2 0, E3 0, E4 0 } C_DIS
LIN{ E6POS: X 756.7952, Y -17.2018, Z -126.0150, A 0, B 90, C 0, E1 0, E2 0, E3 0, E4 0 } C_DIS
LIN{ E6POS: X 755.7975, Y -17.1347, Z -126.0150, A 0, B 90, C 0, E1 0, E2 0, E3 0, E4 0 } C_DIS
LIN{ E6POS: X 754.7998, Y -17.0675, Z -126.0150, A 0, B 90, C 0, E1 0, E2 0, E3 0, E4 0 } C_DIS
LIN{ E6POS: X 754.0056, Y -17.0141, Z -126.0150, A 0, B 90, C 0, E1 0, E2 0, E3 0, E4 0 } C_DIS
LIN{ E6POS: X 753.4305, Y -17.0066, Z -126.0150, A 0, B 90, C 0, E1 0, E2 0, E3 0, E4 0 } C_DIS
LIN{ E6POS: X 752.4307, Y -16.9903, Z -126.0150, A 0, B 90, C 0, E1 0, E2 0, E3 0, E4 0 } C_DIS
LIN{ E6POS: X 751.4308, Y -16.9741, Z -126.0150, A 0, B 90, C 0, E1 0, E2 0, E3 0, E4 0 } C_DIS
LIN{ E6POS: X 750.4309, Y -16.9578, Z -126.0150, A 0, B 90, C 0, E1 0, E2 0, E3 0, E4 0 } C_DIS
LIN{ E6POS: X 749.4311, Y -16.9416, Z -126.0150, A 0, B 90, C 0, E1 0, E2 0, E3 0, E4 0 } C_DIS
LIN{ E6POS: X 748.4312, Y -16.9254, Z -126.0150, A 0, B 90, C 0, E1 0, E2 0, E3 0, E4 0 } C_DIS
LIN{ E6POS: X 747.4313, Y -16.9091, Z -126.0150, A 0, B 90, C 0, E1 0, E2 0, E3 0, E4 0 } C_DIS
LIN{ E6POS: X 746.4315, Y -16.8929, Z -126.0150, A 0, B 90, C 0, E1 0, E2 0, E3 0, E4 0 } C_DIS
LIN{ E6POS: X 746.1736, Y -16.8887, Z -126.0150, A 0, B 90, C 0, E1 0, E2 0, E3 0, E4 0 } C_DIS
LIN{ E6POS: X 745.7127, Y -16.9149, Z -126.0150, A 0, B 90, C 0, E1 0, E2 0, E3 0, E4 0 } C_DIS
LIN{ E6POS: X 744.7137, Y -16.9597, Z -126.0150, A 0, B 90, C 0, E1 0, E2 0, E3 0, E4 0 } C_DIS
LIN{ E6POS: X 743.7147, Y -17.0044, Z -126.0150, A 0, B 90, C 0, E1 0, E2 0, E3 0, E4 0 } C_DIS
LIN{ E6POS: X 742.7157, Y -17.0492, Z -126.0150, A 0, B 90, C 0, E1 0, E2 0, E3 0, E4 0 } C_DIS
